# B&R Automation Studio project TD52 (part 149)

#### OpcHC.st
```iecst
(*******************************************************************************
OpcHC	 Variables read or write to Testbench

This code is confidential AND proprietary to the INNIO Company.
It may NOT be used in any form, or reproduced in any manner, without the express
written permission of the INNIO Company.
Copyright, INNIO Company, 2022

- list addidtional customized IO channels

Customized modifications: -
------------------------

History:
-------
V1.00.0	14.09.2022		Vockenberger	Neu erstellt
V1.01.0	31.05.2023		Vockenberger	Diff-Drucküberwachung Kühler mit Parameter
		28.07.2023		Vockenberger	Struktur von OPC_DI geändert
V1.02.0	20.03.2024		Vockenberger	Heizhaus und V-Kühler Variablen hinzugefügt
V1.03.0	09.01.2025		Gruber St.		cleanUp after change of parameter structure

Instructions FOR use:
--------------------

Outstandings:
------------

*******************************************************************************)

PROGRAM _CYCLIC

	(**Wird von Motor-CPU geschrieben**********************)
	(**REAL**)
	(*Regler*)
	rOpcHC_R[0]	:=	VIS2MM.tCtr_ChCW_LT_In.Y_man;
	rOpcHC_R[1]	:=	VIS2MM.tCtr_ChCW_LT_In.X_min;
	rOpcHC_R[2]	:=	VIS2MM.tCtr_ChCW_LT_In.X_max;
	rOpcHC_R[3]	:=	INT_TO_REAL(VIS2MM.tCtr_ChCW_LT_In.Tune_quality);

	rOpcHC_R[4]	:=	VIS2MM.tCtr_ChCW_HT_In.Y_man;
	rOpcHC_R[5]	:=	VIS2MM.tCtr_ChCW_HT_In.X_min;
	rOpcHC_R[6]	:=	VIS2MM.tCtr_ChCW_HT_In.X_max;
	rOpcHC_R[7]	:=	INT_TO_REAL(VIS2MM.tCtr_ChCW_HT_In.Tune_quality);

	rOpcHC_R[8]		:=	VIS2MM.tCtr_ChCW_HT_LP_In.Y_man;
	rOpcHC_R[9]		:=	VIS2MM.tCtr_ChCW_HT_LP_In.X_min;
	rOpcHC_R[10]	:=	VIS2MM.tCtr_ChCW_HT_LP_In.X_max;
	rOpcHC_R[11]	:=	INT_TO_REAL(VIS2MM.tCtr_ChCW_HT_LP_In.Tune_quality);

	rOpcHC_R[12]	:=	VIS2MM.tCtr_ChCW_HT_HP_In.Y_man;
	rOpcHC_R[13]	:=	VIS2MM.tCtr_ChCW_HT_HP_In.X_min;
	rOpcHC_R[14]	:=	VIS2MM.tCtr_ChCW_HT_HP_In.X_max;
	rOpcHC_R[15]	:=	INT_TO_REAL(VIS2MM.tCtr_ChCW_HT_HP_In.Tune_quality);

	rOpcHC_R[16]	:=	VIS2MM.tCtr_ChCW_LT_LP_In.Y_man;
	rOpcHC_R[17]	:=	VIS2MM.tCtr_ChCW_LT_LP_In.X_min;
	rOpcHC_R[18]	:=	VIS2MM.tCtr_ChCW_LT_LP_In.X_max;
	rOpcHC_R[19]	:=	INT_TO_REAL(VIS2MM.tCtr_ChCW_LT_LP_In.Tune_quality);

	rOpcHC_R[20]	:=	VIS2MM.tCtr_ChCW_LT_HP_In.Y_man;
	rOpcHC_R[21]	:=	VIS2MM.tCtr_ChCW_LT_HP_In.X_min;
	rOpcHC_R[22]	:=	VIS2MM.tCtr_ChCW_LT_HP_In.X_max;
	rOpcHC_R[23]	:=	INT_TO_REAL(VIS2MM.tCtr_ChCW_LT_HP_In.Tune_quality);

	rOpcHC_R[24]	:=	VIS2MM.tCtr_ECW_In.Y_man;
	rOpcHC_R[25]	:=	VIS2MM.tCtr_ECW_In.X_min;
	rOpcHC_R[26]	:=	VIS2MM.tCtr_ECW_In.X_max;
	rOpcHC_R[27]	:=	INT_TO_REAL(VIS2MM.tCtr_ECW_In.Tune_quality);

	rOpcHC_R[28]	:=	VIS2MM.tCtr_OCW_In.Y_man;
	rOpcHC_R[29]	:=	VIS2MM.tCtr_OCW_In.X_min;
	rOpcHC_R[30]	:=	VIS2MM.tCtr_OCW_In.X_max;
	rOpcHC_R[31]	:=	INT_TO_REAL(VIS2MM.tCtr_OCW_In.Tune_quality);

	rOpcHC_R[32]	:=	VIS2MM.tCtr_ChCW_LT_In.Y_set;
	rOpcHC_R[33]	:=	VIS2MM.tCtr_ChCW_HT_In.Y_set;
	rOpcHC_R[34]	:=	VIS2MM.tCtr_ChCW_LT_LP_In.Y_set;
	rOpcHC_R[35]	:=	VIS2MM.tCtr_ChCW_LT_HP_In.Y_set;
	rOpcHC_R[36]	:=	VIS2MM.tCtr_ChCW_HT_LP_In.Y_set;
	rOpcHC_R[37]	:=	VIS2MM.tCtr_ChCW_HT_HP_In.Y_set;
	rOpcHC_R[38]	:=	VIS2MM.tCtr_ECW_In.Y_set;
	rOpcHC_R[39]	:=	VIS2MM.tCtr_OCW_In.Y_set;

	rOpcHC_R[40]	:=	VIS2MM.rCtr_RW_CV_Set;
	rOpcHC_R[41]	:=	VIS2MM.rCtr_RW_HE_Set;
	rOpcHC_R[42]	:=	VIS2MM.rFC_ChCW_LT_PuSet;
	rOpcHC_R[43]	:=	VIS2MM.rFC_ChCW_HT_PuSet;
	rOpcHC_R[44]	:=	VIS2MM.rFC_ChCW_LT_LP_PuSet;
	rOpcHC_R[45]	:=	VIS2MM.rFC_ChCW_LT_HP_PuSet;
	rOpcHC_R[46]	:=	VIS2MM.rFC_ChCW_HT_LP_PuSet;
	rOpcHC_R[47]	:=	VIS2MM.rFC_ChCW_HT_HP_PuSet;
	rOpcHC_R[48]	:=	VIS2MM.rCtr_RW_LT_1_Set;
	rOpcHC_R[49]	:=	VIS2MM.rFC_ECW_PuSet;
	rOpcHC_R[50]	:=	VIS2MM.rFC_OCW_PuSet;

	rOpcHC_R[51]	:=	VIS2MM.rCtr_RW_HT_1_Set;
	rOpcHC_R[52]	:=	VIS2MM.rCtr_RW_LT_2_Set;
	rOpcHC_R[53]	:=	VIS2MM.rCtr_RW_HT_2_Set;
	rOpcHC_R[54]	:=	VIS2MM.rCtr_RW_ECW_1_Set;
	rOpcHC_R[55]	:=	VIS2MM.rCtr_RW_OCW_1_Set;
	rOpcHC_R[56]	:=	VIS2MM.rCtr_RW_ECW_2_Set;
	rOpcHC_R[57]	:=	VIS2MM.rCtr_RW_OCW_2_Set;
	rOpcHC_R[58]	:=	IN_DI.tT_HW_ReBeEng.Ai;

	rOpcHC_R[59]	:=	Para.tCtr_ECW.W_set;
	rOpcHC_R[60]	:=	Para.tCtr_OCW.W_set;
	rOpcHC_R[61]	:= 	Para.tCtr_ChCW_LT.W_set;
	rOpcHC_R[62]	:=	Para.tCtr_ChCW_LT_LP.W_set;
	rOpcHC_R[63]	:=	Para.tCtr_ChCW_LT_HP.W_set;
	rOpcHC_R[64]	:=	Para.tCtr_ChCW_HT.W_set;
	rOpcHC_R[65]	:=	Para.tCtr_ChCW_HT_LP.W_set;
	rOpcHC_R[66]	:=	Para.tCtr_ChCW_HT_HP.W_set;

	rOpcHC_R[67]	:=	Para.tCtr_ECW.W_min;
	rOpcHC_R[68]	:=	Para.tCtr_ECW.W_max;
	rOpcHC_R[69]	:=	Para.tCtr_ECW.Y_min;
	rOpcHC_R[70]	:=	Para.tCtr_ECW.Y_max;
	rOpcHC_R[71]	:=	Para.tCtr_OCW.W_min;
	rOpcHC_R[72]	:=	Para.tCtr_OCW.W_max;
	rOpcHC_R[73]	:=	Para.tCtr_OCW.Y_min;
	rOpcHC_R[74]	:=	Para.tCtr_OCW.Y_max;

	rOpcHC_R[75]	:=	Para.tCtr_ChCW_LT.W_min;
	rOpcHC_R[76]	:=	Para.tCtr_ChCW_LT.W_max;
	rOpcHC_R[77]	:=	Para.tCtr_ChCW_LT.Y_min;
	rOpcHC_R[78]	:=	Para.tCtr_ChCW_LT.Y_max;
	rOpcHC_R[79]	:=	Para.tCtr_ChCW_LT_LP.W_min;
	rOpcHC_R[80]	:=	Para.tCtr_ChCW_LT_LP.W_max;
	rOpcHC_R[81]	:=	Para.tCtr_ChCW_LT_LP.Y_min;
	rOpcHC_R[82]	:=	Para.tCtr_ChCW_LT_LP.Y_max;

	rOpcHC_R[83]	:=	Para.tCtr_ChCW_LT_HP.W_min;
	rOpcHC_R[84]	:=	Para.tCtr_ChCW_LT_HP.W_max;
	rOpcHC_R[85]	:=	Para.tCtr_ChCW_LT_HP.Y_min;
	rOpcHC_R[86]	:=	Para.tCtr_ChCW_LT_HP.Y_max;
	rOpcHC_R[87]	:=	Para.tCtr_ChCW_HT.W_min;
	rOpcHC_R[88]	:=	Para.tCtr_ChCW_HT.W_max;
	rOpcHC_R[89]	:=	Para.tCtr_ChCW_HT.Y_min;
	rOpcHC_R[90]	:=	Para.tCtr_ChCW_HT.Y_max;

	rOpcHC_R[91]	:=	Para.tCtr_ChCW_HT_LP.W_min;
	rOpcHC_R[92]	:=	Para.tCtr_ChCW_HT_LP.W_max;
	rOpcHC_R[93]	:=	Para.tCtr_ChCW_HT_LP.Y_min;
	rOpcHC_R[94]	:=	Para.tCtr_ChCW_HT_LP.Y_max;
	rOpcHC_R[95]	:=	Para.tCtr_ChCW_HT_HP.W_min;
	rOpcHC_R[96]	:=	Para.tCtr_ChCW_HT_HP.W_max;
	rOpcHC_R[97]	:=	Para.tCtr_ChCW_HT_HP.Y_min;
	rOpcHC_R[98]	:=	Para.tCtr_ChCW_HT_HP.Y_max;

	rOpcHC_R[99]	:=	VIS2MM.tPreHeatWDayLT[0].Hour;
	rOpcHC_R[100]	:=	VIS2MM.tPreHeatWDayLT[0].Minute;
	rOpcHC_R[101]	:=	VIS2MM.tPreHeatWDayLT[1].Hour;
	rOpcHC_R[102]	:=	VIS2MM.tPreHeatWDayLT[1].Minute;
	rOpcHC_R[103]	:=	VIS2MM.tPreHeatWDayLT[2].Hour;
	rOpcHC_R[104]	:=	VIS2MM.tPreHeatWDayLT[2].Minute;
	rOpcHC_R[105]	:=	VIS2MM.tPreHeatWDayLT[3].Hour;
	rOpcHC_R[106]	:=	VIS2MM.tPreHeatWDayLT[3].Minute;
	rOpcHC_R[107]	:=	VIS2MM.tPreHeatWDayLT[4].Hour;
	rOpcHC_R[108]	:=	VIS2MM.tPreHeatWDayLT[4].Minute;
	rOpcHC_R[109]	:=	VIS2MM.tPreHeatWDayLT[5].Hour;
	rOpcHC_R[110]	:=	VIS2MM.tPreHeatWDayLT[5].Minute;
	rOpcHC_R[111]	:=	VIS2MM.tPreHeatWDayLT[6].Hour;
	rOpcHC_R[112]	:=	VIS2MM.tPreHeatWDayLT[6].Minute;

	rOpcHC_R[113]	:=	VIS2MM.rT_LT_HP_Preh;
	rOpcHC_R[114]	:=	VIS2MM.rT_LT_LP_Preh;

	rOpcHC_R[115]	:=	IN_DI.tT_Ch_T2LP_A.Ai;
	rOpcHC_R[116]	:=	IN_DI.tT_Ch_T2LP_B.Ai;

	(**BOOL**)
	bOpcHC_R[0]  := VIS2MM.tCtr_ChCW_LT_In.Y_man_Active;
	bOpcHC_R[1]  := VIS2MM.tCtr_ChCW_LT_In.W_ext_Active;
	bOpcHC_R[2]  := VIS2MM.tCtr_ChCW_LT_In.Tune_PI;
	bOpcHC_R[3]  := VIS2MM.tCtr_ChCW_LT_In.Tune_PID;
	bOpcHC_R[4]  := VIS2MM.tCtr_ChCW_LT_In.Tune_start;
	bOpcHC_R[5]  := VIS2MM.tCtr_ChCW_LT_In.Tune_stop;
	bOpcHC_R[6]  := VIS2MM.tCtr_ChCW_LT_In.Tune_takeover;
	bOpcHC_R[7]	 := VIS2MM.tCtr_ChCW_LT_In.W_set2_Active;

	bOpcHC_R[8]   := VIS2MM.tCtr_ChCW_HT_In.Y_man_Active;
	bOpcHC_R[9]   := VIS2MM.tCtr_ChCW_HT_In.W_ext_Active;
	bOpcHC_R[10]  := VIS2MM.tCtr_ChCW_HT_In.Tune_PI;
	bOpcHC_R[11]  := VIS2MM.tCtr_ChCW_HT_In.Tune_PID;
	bOpcHC_R[12]  := VIS2MM.tCtr_ChCW_HT_In.Tune_start;
	bOpcHC_R[13]  := VIS2MM.tCtr_ChCW_HT_In.Tune_stop;
	bOpcHC_R[14]  := VIS2MM.tCtr_ChCW_HT_In.Tune_takeover;
	bOpcHC_R[15]  := VIS2MM.tCtr_ChCW_HT_In.W_set2_Active;

	bOpcHC_R[16]  := VIS2MM.tCtr_ChCW_HT_LP_In.Y_man_Active;
	bOpcHC_R[17]  := VIS2MM.tCtr_ChCW_HT_LP_In.W_ext_Active;
	bOpcHC_R[18]  := VIS2MM.tCtr_ChCW_HT_LP_In.Tune_PI;
	bOpcHC_R[19]  := VIS2MM.tCtr_ChCW_HT_LP_In.Tune_PID;
	bOpcHC_R[20]  := VIS2MM.tCtr_ChCW_HT_LP_In.Tune_start;
	bOpcHC_R[21]  := VIS2MM.tCtr_ChCW_HT_LP_In.Tune_stop;
	bOpcHC_R[22]  := VIS2MM.tCtr_ChCW_HT_LP_In.Tune_takeover;
	bOpcHC_R[23]  := VIS2MM.tCtr_ChCW_HT_LP_In.W_set2_Active;

	bOpcHC_R[24]  := VIS2MM.tCtr_ChCW_HT_HP_In.Y_man_Active;
	bOpcHC_R[25]  := VIS2MM.tCtr_ChCW_HT_HP_In.W_ext_Active;
	bOpcHC_R[26]  := VIS2MM.tCtr_ChCW_HT_HP_In.Tune_PI;
	bOpcHC_R[27]  := VIS2MM.tCtr_ChCW_HT_HP_In.Tune_PID;
	bOpcHC_R[28]  := VIS2MM.tCtr_ChCW_HT_HP_In.Tune_start;
	bOpcHC_R[29]  := VIS2MM.tCtr_ChCW_HT_HP_In.Tune_stop;
	bOpcHC_R[30]  := VIS2MM.tCtr_ChCW_HT_HP_In.Tune_takeover;
	bOpcHC_R[31]  := VIS2MM.tCtr_ChCW_HT_HP_In.W_set2_Active;

	bOpcHC_R[32]  := VIS2MM.tCtr_ChCW_LT_LP_In.Y_man_Active;
	bOpcHC_R[33]  := VIS2MM.tCtr_ChCW_LT_LP_In.W_ext_Active;
	bOpcHC_R[34]  := VIS2MM.tCtr_ChCW_LT_LP_In.Tune_PI;
	bOpcHC_R[35]  := VIS2MM.tCtr_ChCW_LT_LP_In.Tune_PID;
	bOpcHC_R[36]  := VIS2MM.tCtr_ChCW_LT_LP_In.Tune_start;
	bOpcHC_R[37]  := VIS2MM.tCtr_ChCW_LT_LP_In.Tune_stop;
	bOpcHC_R[38]  := VIS2MM.tCtr_ChCW_LT_LP_In.Tune_takeover;
	bOpcHC_R[39]  := VIS2MM.tCtr_ChCW_LT_LP_In.W_set2_Active;

	bOpcHC_R[40]  := VIS2MM.tCtr_ChCW_LT_HP_In.Y_man_Active;
	bOpcHC_R[41]  := VIS2MM.tCtr_ChCW_LT_HP_In.W_ext_Active;
	bOpcHC_R[42]  := VIS2MM.tCtr_ChCW_LT_HP_In.Tune_PI;
	bOpcHC_R[43]  := VIS2MM.tCtr_ChCW_LT_HP_In.Tune_PID;
	bOpcHC_R[44]  := VIS2MM.tCtr_ChCW_LT_HP_In.Tune_start;
	bOpcHC_R[45]  := VIS2MM.tCtr_ChCW_LT_HP_In.Tune_stop;
	bOpcHC_R[46]  := VIS2MM.tCtr_ChCW_LT_HP_In.Tune_takeover;
	bOpcHC_R[47]  := VIS2MM.tCtr_ChCW_LT_HP_In.W_set2_Active;

	bOpcHC_R[48]  := VIS2MM.tCtr_ECW_In.Y_man_Active;
	bOpcHC_R[49]  := VIS2MM.tCtr_ECW_In.W_ext_Active;
	bOpcHC_R[50]  := VIS2MM.tCtr_ECW_In.Tune_PI;
	bOpcHC_R[51]  := VIS2MM.tCtr_ECW_In.Tune_PID;
	bOpcHC_R[52]  := VIS2MM.tCtr_ECW_In.Tune_start;
	bOpcHC_R[53]  := VIS2MM.tCtr_ECW_In.Tune_stop;
	bOpcHC_R[54]  := VIS2MM.tCtr_ECW_In.Tune_takeover;
	bOpcHC_R[55]  := VIS2MM.tCtr_ECW_In.W_set2_Active;

	bOpcHC_R[56]  := VIS2MM.tCtr_OCW_In.Y_man_Active;
	bOpcHC_R[57]  := VIS2MM.tCtr_OCW_In.W_ext_Active;
	bOpcHC_R[58]  := VIS2MM.tCtr_OCW_In.Tune_PI;
	bOpcHC_R[59]  := VIS2MM.tCtr_OCW_In.Tune_PID;
	bOpcHC_R[60]  := VIS2MM.tCtr_OCW_In.Tune_start;
	bOpcHC_R[61]  := VIS2MM.tCtr_OCW_In.Tune_stop;
	bOpcHC_R[62]  := VIS2MM.tCtr_OCW_In.Tune_takeover;
	bOpcHC_R[63]  := VIS2MM.tCtr_OCW_In.W_set2_Active;

	bOpcHC_R[64]  := bCtr_LT_In_Y_set_Active;
	bOpcHC_R[65]  := bCtr_HT_In_Y_set_Active;
	bOpcHC_R[66]  := bCtr_LT_LP_In_Y_set_Active;
	bOpcHC_R[67]  := bCtr_LT_HP_In_Y_set_Active;
	bOpcHC_R[68]  := bCtr_HT_LP_In_Y_set_Active;
	bOpcHC_R[69]  := bCtr_HT_HP_In_Y_set_Active;
	bOpcHC_R[70]  := bCtr_ECW_In_Y_set_Active;
	bOpcHC_R[71]  := bCtr_OCW_In_Y_set_Active;

	bOpcHC_R[72]  := VIS2MM.bMan_ECW_Pump;
	bOpcHC_R[73]  := VIS2MM.bMan_OCW_Pump;
	bOpcHC_R[74]  := VIS2MM.bMan_LT_Pump;
	bOpcHC_R[75]  := VIS2MM.bMan_HT_Pump;
	bOpcHC_R[76]  := VIS2MM.bMan_LT_LP_Pump;
	bOpcHC_R[77]  := VIS2MM.bMan_LT_HP_Pump;
	bOpcHC_R[78]  := VIS2MM.bMan_HT_LP_Pump;
	bOpcHC_R[79]  := VIS2MM.bMan_HT_HP_Pump;

	bOpcHC_R[80]	:=	VIS2MM.bMan_BoilerHouse_Pump;
	bOpcHC_R[81]	:=	VIS2MM.bMan_SecCirc_Pump;
	bOpcHC_R[82]	:=	VIS2MM.bPreHeatWDayLT_CtrActive;
	bOpcHC_R[83]	:=	VIS2MM.bLT_PreH_Dem;
	bOpcHC_R[84]	:=	VIS2MM.tPreHeatWDayLT[0].Active;
	bOpcHC_R[85]	:=	VIS2MM.tPreHeatWDayLT[1].Active;
	bOpcHC_R[86]	:=	VIS2MM.tPreHeatWDayLT[2].Active;
	bOpcHC_R[87]	:=	VIS2MM.tPreHeatWDayLT[3].Active;
	bOpcHC_R[88]	:=	VIS2MM.tPreHeatWDayLT[4].Active;
	bOpcHC_R[89]	:=	VIS2MM.tPreHeatWDayLT[5].Active;
	bOpcHC_R[90]	:=	VIS2MM.tPreHeatWDayLT[6].Active;
	bOpcHC_R[91]	:=	VIS2MM.tPreHeatWDayLT[7].Active;
	bOpcHC_R[92]	:=	VIS2MM.tPreHeatWDayLT[0].Off;
	bOpcHC_R[93]	:=	VIS2MM.tPreHeatWDayLT[1].Off;
	bOpcHC_R[94]	:=	VIS2MM.tPreHeatWDayLT[2].Off;
	bOpcHC_R[95]	:=	VIS2MM.tPreHeatWDayLT[3].Off;
	bOpcHC_R[96]	:=	VIS2MM.tPreHeatWDayLT[4].Off;
	bOpcHC_R[97]	:=	VIS2MM.tPreHeatWDayLT[5].Off;
	bOpcHC_R[98]	:=	VIS2MM.tPreHeatWDayLT[6].Off;
	bOpcHC_R[99]	:=	IN_DI.tT_Ch_T2LP_A.Exist;
	bOpcHC_R[100];

	(**Wird von Prüfstands-CPU geschrieben**********************)
	(**REAL**)
	MM2VIS.rT_ChCW_Re_LT		:=	rOpcHC_W[0];
	MM2VIS.rPr_ChCW_Re_LT		:=	rOpcHC_W[1];
	MM2VIS.rT_ChCW_Su_LT		:=	rOpcHC_W[2];
	MM2VIS.rPr_ChCW_Su_LT		:=	rOpcHC_W[3];
	MM2VIS.rT_ChCW_Re_HT		:=	rOpcHC_W[4];
	MM2VIS.rPr_ChCW_Re_HT		:=	rOpcHC_W[5];
	MM2VIS.rT_ChCW_Su_HT		:=	rOpcHC_W[6];
	MM2VIS.rPr_ChCW_Su_HT		:=	rOpcHC_W[7];
	MM2VIS.rT_ChCW_Re_HT_LP		:=	rOpcHC_W[8];
	MM2VIS.rPr_ChCW_Re_HT_LP	:=	rOpcHC_W[9];

	MM2VIS.rT_ChCW_Re_HT_HP		:=	rOpcHC_W[10];
	MM2VIS.rPr_ChCW_Re_HT_HP	:=	rOpcHC_W[11];
	MM2VIS.rT_ChCW_Su_HT_LP		:=	rOpcHC_W[12];
	MM2VIS.rPr_ChCW_Su_HT_LP	:=	rOpcHC_W[13];
	MM2VIS.rT_ChCW_Su_HT_HP		:=	rOpcHC_W[14];
	MM2VIS.rPr_ChCW_Su_HT_HP	:=	rOpcHC_W[15];
	MM2VIS.rT_ChCW_Re_LT_LP		:=	rOpcHC_W[16];
	MM2VIS.rPr_ChCW_Re_LT_LP	:=	rOpcHC_W[17];
	MM2VIS.rT_ChCW_Re_LT_HP		:=	rOpcHC_W[18];
	MM2VIS.rPr_ChCW_Re_LT_HP	:=	rOpcHC_W[19];

	MM2VIS.rT_ChCW_Su_LT_LP		:=	rOpcHC_W[20];
	MM2VIS.rPr_ChCW_Su_LT_LP	:=	rOpcHC_W[21];
	MM2VIS.rT_ChCW_Su_LT_HP		:=	rOpcHC_W[22];
	MM2VIS.rPr_ChCW_Su_LT_HP	:=	rOpcHC_W[23];
	MM2VIS.rT_OCW_Re			:=	rOpcHC_W[24];
	MM2VIS.rPr_OCW_Re			:=	rOpcHC_W[25];
	MM2VIS.rT_OCW_Su			:=	rOpcHC_W[26];
	MM2VIS.rPr_OCW_Su			:=	rOpcHC_W[27];
	MM2VIS.rT_ECW_Re			:=	rOpcHC_W[28];
	MM2VIS.rPr_ECW_Re			:=	rOpcHC_W[29];

	MM2VIS.rT_ECW_Su			:=	rOpcHC_W[30];
	MM2VIS.rPr_ECW_Su			:=	rOpcHC_W[31];
	MM2VIS.rVol_ChCW_Re_LT		:=	rOpcHC_W[32];
	MM2VIS.rVol_ChCW_Su_LT		:=	rOpcHC_W[33];
	MM2VIS.rVol_ChCW_Re_HT		:=	rOpcHC_W[34];
	MM2VIS.rVol_ChCW_Su_HT		:=	rOpcHC_W[35];
	MM2VIS.rVol_ChCW_Re_HT_LP	:=	rOpcHC_W[36];
	MM2VIS.rVol_ChCW_Su_HT_LP	:=	rOpcHC_W[37];
	MM2VIS.rVol_ChCW_Re_HT_HP	:=	rOpcHC_W[38];
	MM2VIS.rVol_ChCW_Su_HT_HP	:=	rOpcHC_W[39];

	MM2VIS.rVol_ChCW_Re_LT_LP	:=	rOpcHC_W[40];
	MM2VIS.rVol_ChCW_Su_LT_LP	:=	rOpcHC_W[41];
	MM2VIS.rVol_ChCW_Re_LT_HP	:=	rOpcHC_W[42];
	MM2VIS.rVol_ChCW_Su_LT_HP	:=	rOpcHC_W[43];
	MM2VIS.rVol_ECW_Re			:=	rOpcHC_W[44];
	MM2VIS.rVol_ECW_Su			:=	rOpcHC_W[45];
	MM2VIS.rVol_OCW_Re			:=	rOpcHC_W[46];
	MM2VIS.rVol_OCW_Su			:=	rOpcHC_W[47];
	MM2VIS.rPosAct_RW_LT_1		:=	rOpcHC_W[48];
	MM2VIS.rPosAct_RW_HT_1		:=	rOpcHC_W[49];

	MM2VIS.rT_ChCW_LT_IC_Re		:=	rOpcHC_W[50];
	MM2VIS.rPr_ChCW_LT_IC_Re	:=	rOpcHC_W[51];
	MM2VIS.rT_ChCW_HT_IC_Re		:=	rOpcHC_W[52];
	MM2VIS.rPr_ChCW_HT_IC_Re	:=	rOpcHC_W[53];
	MM2VIS.rT_ChCW_LT_LP_IC_Re	:=	rOpcHC_W[54];
	MM2VIS.rPr_ChCW_LT_LP_IC_Re	:=	rOpcHC_W[55];
	MM2VIS.rT_ChCW_LT_HP_IC_Re	:=	rOpcHC_W[56];
	MM2VIS.rPr_ChCW_LT_HP_IC_Re	:=	rOpcHC_W[57];
	MM2VIS.rT_ChCW_HT_LP_IC_Re	:=	rOpcHC_W[58];
	MM2VIS.rPr_ChCW_HT_LP_IC_Re	:=	rOpcHC_W[59];

	MM2VIS.rT_ChCW_HT_HP_IC_Re	:=	rOpcHC_W[60];
	MM2VIS.rPr_ChCW_HT_HP_IC_Re	:=	rOpcHC_W[61];
	MM2VIS.rT_RW_Re				:=	rOpcHC_W[62];
	MM2VIS.rT_RW_Su				:=	rOpcHC_W[63];
	MM2VIS.rT_ECW_IC_Re			:=	rOpcHC_W[64];
	MM2VIS.rPr_ECW_IC_Re		:=	rOpcHC_W[65];
	MM2VIS.rT_OCW_IC_Re			:=	rOpcHC_W[66];
	MM2VIS.rPr_OCW_IC_Re		:=	rOpcHC_W[67];
	MM2VIS.rT_ChCW_LT_IC_Su		:=	rOpcHC_W[68];
	MM2VIS.rPr_ChCW_LT_IC_Su	:=	rOpcHC_W[69];

	MM2VIS.rT_ChCW_HT_IC_Su		:=	rOpcHC_W[70];
	MM2VIS.rPr_ChCW_HT_IC_Su	:=	rOpcHC_W[71];
	MM2VIS.rT_ChCW_LT_LP_IC_Su	:=	rOpcHC_W[72];
	MM2VIS.rPr_ChCW_LT_LP_IC_Su	:=	rOpcHC_W[73];
	MM2VIS.rT_ChCW_LT_HP_IC_Su	:=	rOpcHC_W[74];
	MM2VIS.rPr_ChCW_LT_HP_IC_Su	:=	rOpcHC_W[75];
	MM2VIS.rT_ChCW_HT_LP_IC_Su	:=	rOpcHC_W[76];
	MM2VIS.rPr_ChCW_HT_LP_IC_Su	:=	rOpcHC_W[77];
	MM2VIS.rT_ChCW_HT_HP_IC_Su	:=	rOpcHC_W[78];
	MM2VIS.rPr_ChCW_HT_HP_IC_Su	:=	rOpcHC_W[79];

	MM2VIS.rPr_RW_LT_Re_1		:=	rOpcHC_W[80];
	MM2VIS.rPr_RW_LT_Su_1		:=	rOpcHC_W[81];
	MM2VIS.rT_ECW_IC_Su			:=	rOpcHC_W[82];
	MM2VIS.rPr_ECW_IC_Su		:=	rOpcHC_W[83];
	MM2VIS.rT_OCW_IC_Su			:=	rOpcHC_W[84];
	MM2VIS.rPr_OCW_IC_Su		:=	rOpcHC_W[85];
	MM2VIS.rT_Cooler_ChCW_LT_Re_1	:=	rOpcHC_W[86];
	MM2VIS.rT_Cooler_ChCW_HT_Re_1	:=	rOpcHC_W[87];
	MM2VIS.rT_Cooler_ChCW_HT_Re_3	:=	rOpcHC_W[88];
	MM2VIS.rT_Cooler_ChCW_HT_Re_4	:=	rOpcHC_W[89];

	MM2VIS.rT_Cooler_ChCW_HT_Re_5	:=	rOpcHC_W[90];
	MM2VIS.rT_Cooler_ChCW_HT_Su_3	:=	rOpcHC_W[91];
	MM2VIS.rT_Cooler_ChCW_LT_Re_2		:=	rOpcHC_W[92];
	MM2VIS.rT_Cooler_ChCW_HT_Re_2		:=	rOpcHC_W[93];
	MM2VIS.rT_Cooler_ChCW_HT_Su_4	:=	rOpcHC_W[94];
	MM2VIS.rT_Cooler_ChCW_HT_Su_5	:=	rOpcHC_W[95];
	MM2VIS.rT_CoolerCabinet_HT_1	:=	rOpcHC_W[96];
	MM2VIS.rT_CoolerCabinet_HT_2	:=	rOpcHC_W[97];
	MM2VIS.rPr_Cooler_ChCW_LT_Re_1		:=	rOpcHC_W[98];
	MM2VIS.rPr_Cooler_ChCW_HT_Re_1		:=	rOpcHC_W[99];

	MM2VIS.rT_CoolerCabinet_HT_3		:=	rOpcHC_W[100];
	MM2VIS.rT_CoolerCabinet_HT_4		:=	rOpcHC_W[101];
	MM2VIS.rT_CoolerCabinet_HT_5		:=	rOpcHC_W[102];
	MM2VIS.rT_Cooler_OCW_Re_3			:=	rOpcHC_W[103];
	MM2VIS.rPr_Cooler_ChCW_LT_Re_2		:=	rOpcHC_W[104];
	MM2VIS.rPr_Cooler_ChCW_HT_Re_2		:=	rOpcHC_W[105];
	MM2VIS.rT_Cooler_OCW_Su_3			:=	rOpcHC_W[106];
	MM2VIS.rT_CoolerCabinet_OCW_1		:=	rOpcHC_W[107];
	MM2VIS.rT_CoolerCabinet_OCW_2		:=	rOpcHC_W[108];
	MM2VIS.rT_CoolerCabinet_OCW_3		:=	rOpcHC_W[109];

	MM2VIS.rT_Cooler_ChCW_LT_Su_1		:=	rOpcHC_W[110];
	MM2VIS.rT_Cooler_ChCW_HT_Su_1		:=	rOpcHC_W[111];
	MM2VIS.rT_Cooler_ECW_Re_3			:=	rOpcHC_W[112];
	MM2VIS.rT_Cooler_ECW_Re_4			:=	rOpcHC_W[113];
	MM2VIS.rT_Cooler_ECW_Su_3			:=	rOpcHC_W[114];
	MM2VIS.rT_Cooler_ECW_Su_4			:=	rOpcHC_W[115];
	MM2VIS.rT_Cooler_ChCW_LT_Su_2		:=	rOpcHC_W[116];
	MM2VIS.rT_Cooler_ChCW_HT_Su_2		:=	rOpcHC_W[117];
	MM2VIS.rT_CoolerCabinet_ECW_1		:=	rOpcHC_W[118];
	MM2VIS.rT_CoolerCabinet_ECW_2		:=	rOpcHC_W[119];

	MM2VIS.rT_CoolerCabinet_ECW_3		:=	rOpcHC_W[120];
	MM2VIS.rT_CoolerCabinet_ECW_4		:=	rOpcHC_W[121];
	MM2VIS.rPr_Cooler_ChCW_LT_Su_1		:=	rOpcHC_W[122];
	MM2VIS.rPr_Cooler_ChCW_HT_Su_1		:=	rOpcHC_W[123];
	MM2VIS.rT_Cooler_ChCW_LT_Re_3		:=	rOpcHC_W[124];
	MM2VIS.rT_Cooler_ChCW_LT_Re_4		:=	rOpcHC_W[125];
	MM2VIS.rT_Cooler_ChCW_LT_Re_5		:=	rOpcHC_W[126];
	MM2VIS.rT_Cooler_ChCW_LT_Su_3		:=	rOpcHC_W[127];
	MM2VIS.rPr_Cooler_ChCW_LT_Su_2		:=	rOpcHC_W[128];
	MM2VIS.rPr_Cooler_ChCW_HT_Su_2		:=	rOpcHC_W[129];

	MM2VIS.rT_Cooler_ChCW_LT_Su_4	:=	rOpcHC_W[130];
	MM2VIS.rT_Cooler_ChCW_LT_Su_5	:=	rOpcHC_W[131];
	MM2VIS.rT_CoolerCabinet_LT_1	:=	rOpcHC_W[132];
	MM2VIS.rT_CoolerCabinet_LT_2	:=	rOpcHC_W[133];
	MM2VIS.rPr_RW_LT_Re_2		:=	rOpcHC_W[134];
	MM2VIS.rPr_RW_LT_Su_2		:=	rOpcHC_W[135];
	MM2VIS.rT_Cooler_ECW_Re_1	:=	rOpcHC_W[136];
	MM2VIS.rT_Cooler_ECW_Re_2	:=	rOpcHC_W[137];
	MM2VIS.rT_Cooler_OCW_Re_1	:=	rOpcHC_W[138];
	MM2VIS.rT_Cooler_OCW_Re_2	:=	rOpcHC_W[139];

	MM2VIS.rPr_RW_HT_Re_1		:=	rOpcHC_W[140];
	MM2VIS.rPr_RW_HT_Su_1		:=	rOpcHC_W[141];
	MM2VIS.rT_Cooler_ECW_Su_1	:=	rOpcHC_W[142];
	MM2VIS.rT_Cooler_ECW_Su_2	:=	rOpcHC_W[143];
	MM2VIS.rT_Cooler_OCW_Su_1	:=	rOpcHC_W[144];
	MM2VIS.rT_Cooler_OCW_Su_2	:=	rOpcHC_W[145];
	MM2VIS.rT_ChCW_LT_bCV		:=	rOpcHC_W[146];
	MM2VIS.rT_RW_HE_Re			:=	rOpcHC_W[147];
	MM2VIS.rT_RW_HE_Su			:=	rOpcHC_W[148];
	MM2VIS.rPr_RW_HT_Re_2		:=	rOpcHC_W[149];

	MM2VIS.rPr_RW_HT_Su_2		:=	rOpcHC_W[150];
	MM2VIS.rPr_Cooler_ECW_Re_1	:=	rOpcHC_W[151];
	MM2VIS.rPr_Cooler_ECW_Re_2	:=	rOpcHC_W[152];
	MM2VIS.rPr_Cooler_OCW_Re_1	:=	rOpcHC_W[153];
	MM2VIS.rPr_Cooler_OCW_Re_2	:=	rOpcHC_W[154];
	MM2VIS.rPr_RW_ECW_Re_1		:=	rOpcHC_W[155];
	MM2VIS.rPr_RW_ECW_Su_1		:=	rOpcHC_W[156];
	MM2VIS.rPr_Cooler_ECW_Su_1	:=	rOpcHC_W[157];
	MM2VIS.rPr_Cooler_ECW_Su_2	:=	rOpcHC_W[158];
	MM2VIS.rPr_Cooler_OCW_Su_1	:=	rOpcHC_W[159];

	MM2VIS.rPr_Cooler_OCW_Su_2	:=	rOpcHC_W[160];
	MM2VIS.rPr_RW_HE_Re			:=	rOpcHC_W[161];
	MM2VIS.rPr_RW_HE_Su			:=	rOpcHC_W[162];
	MM2VIS.rFC_ChCW_LT_Pump		:=	rOpcHC_W[163];
	MM2VIS.rFC_ChCW_HT_Pump		:=	rOpcHC_W[164];
	MM2VIS.rFC_ChCW_LT_LP_Pump	:=	rOpcHC_W[165];
	MM2VIS.rFC_ChCW_LT_HP_Pump	:=	rOpcHC_W[166];
	MM2VIS.rFC_ChCW_HT_LP_Pump	:=	rOpcHC_W[167];
	MM2VIS.rFC_ChCW_HT_HP_Pump	:=	rOpcHC_W[168];
	MM2VIS.rPr_RW_ECW_Re_2		:=	rOpcHC_W[169];

	MM2VIS.rFC_ECW_Pump			:=	rOpcHC_W[170];
	MM2VIS.rFC_OCW_Pump			:=	rOpcHC_W[171];
	MM2VIS.rFC_ChCW_LT_Cooler_1	:=	rOpcHC_W[172];
	MM2VIS.rFC_ChCW_HT_Cooler_1	:=	rOpcHC_W[173];
	MM2VIS.rT_CoolerCabinet_LT_3	:=	rOpcHC_W[174];
	MM2VIS.rT_CoolerCabinet_LT_4	:=	rOpcHC_W[175];
	MM2VIS.rT_CoolerCabinet_LT_5	:=	rOpcHC_W[176];
	MM2VIS.rFC_ChCW_HT_HP_Cooler_1	:=	rOpcHC_W[177];
	MM2VIS.rFC_ChCW_LT_Cooler_2	:=	rOpcHC_W[178];
	MM2VIS.rFC_ChCW_HT_Cooler_2	:=	rOpcHC_W[179];

	MM2VIS.rFC_ChCW_LT_LP_Cooler_2	:=	rOpcHC_W[180];
	MM2VIS.rFC_ChCW_LT_HP_Cooler_2	:=	rOpcHC_W[181];
	MM2VIS.rFC_ChCW_HT_LP_Cooler_2	:=	rOpcHC_W[182];
	MM2VIS.rFC_ChCW_HT_HP_Cooler_2	:=	rOpcHC_W[183];
	MM2VIS.rPr_RW_ECW_Su_2		:=	rOpcHC_W[184];
	MM2VIS.rFC_ECW_Cooler_1		:=	rOpcHC_W[185];
	MM2VIS.rFC_OCW_Cooler_1		:=	rOpcHC_W[186];
	MM2VIS.rPr_RW_OCW_Re_1		:=	rOpcHC_W[187];
	MM2VIS.rFC_ECW_Cooler_2		:=	rOpcHC_W[188];
	MM2VIS.rFC_OCW_Cooler_2		:=	rOpcHC_W[189];

	MM2VIS.rT_ChCW_LT_LP_bCV	:=	rOpcHC_W[190];
	MM2VIS.rT_ChCW_LT_HP_bCV	:=	rOpcHC_W[191];
	MM2VIS.rT_ChCW_HT_bCV		:=	rOpcHC_W[192];
	MM2VIS.rT_ChCW_HT_LP_bCV	:=	rOpcHC_W[193];
	MM2VIS.rT_ChCW_HT_HP_bCV	:=	rOpcHC_W[194];
	MM2VIS.rPr_RW_OCW_Su_1		:=	rOpcHC_W[195];
	MM2VIS.rT_ECW_bCV			:=	rOpcHC_W[196];
	MM2VIS.rT_OCW_bCV			:=	rOpcHC_W[197];
	MM2VIS.rPosAct_ChCW_LT		:=	rOpcHC_W[198];
	MM2VIS.rPosAct_ChCW_HT		:=	rOpcHC_W[199];

	MM2VIS.rPosAct_ChCW_HT_LP	:=	rOpcHC_W[200];
	MM2VIS.rPosAct_ChCW_HT_HP	:=	rOpcHC_W[201];
	MM2VIS.rPosAct_ChCW_LT_LP	:=	rOpcHC_W[202];
	MM2VIS.rPosAct_ChCW_LT_HP	:=	rOpcHC_W[203];
	MM2VIS.rPosAct_ECW			:=	rOpcHC_W[204];
	MM2VIS.rPosAct_OCW			:=	rOpcHC_W[205];
	MM2VIS.rPr_RW_OCW_Re_2		:=	rOpcHC_W[206];
	MM2VIS.rPosAct_RW_CV		:=	rOpcHC_W[207];
	MM2VIS.rPosAct_RW_HE		:=	rOpcHC_W[208];

	(**Regler**)
	MM2VIS.rCtr_ChCW_LT_In_X		:=	rOpcHC_W[209];
	MM2VIS.tCtr_ChCW_LT_Out.Y		:=	rOpcHC_W[210];
	MM2VIS.tCtr_ChCW_LT_Out.Y_min_act	:=	rOpcHC_W[211];
	MM2VIS.tCtr_ChCW_LT_Out.Y_max_act	:=	rOpcHC_W[212];
	MM2VIS.tCtr_ChCW_LT_Out.W		:=	rOpcHC_W[213];
	MM2VIS.tCtr_ChCW_LT_Out.e		:=	rOpcHC_W[214];
	MM2VIS.tCtr_ChCW_LT_Out.Kp_tune	:=	rOpcHC_W[215];
	MM2VIS.tCtr_ChCW_LT_Out.Tn_tune	:=	rOpcHC_W[216];
	MM2VIS.tCtr_ChCW_LT_Out.Tv_tune	:=	rOpcHC_W[217];
	MM2VIS.tCtr_ChCW_LT_Out.status	:=	REAL_TO_UINT(rOpcHC_W[218]);
	MM2VIS.tCtr_ChCW_LT_Out.Kp_act	:=	rOpcHC_W[219];
	MM2VIS.tCtr_ChCW_LT_Out.Tn_act	:=	rOpcHC_W[220];
	MM2VIS.tCtr_ChCW_LT_Out.Tv_act	:=	rOpcHC_W[221];

	MM2VIS.rCtr_ChCW_HT_In_X		:=	rOpcHC_W[222];
	MM2VIS.tCtr_ChCW_HT_Out.Y		:=	rOpcHC_W[223];
	MM2VIS.tCtr_ChCW_HT_Out.Y_min_act	:=	rOpcHC_W[224];
	MM2VIS.tCtr_ChCW_HT_Out.Y_max_act	:=	rOpcHC_W[225];
	MM2VIS.tCtr_ChCW_HT_Out.W		:=	rOpcHC_W[226];
	MM2VIS.tCtr_ChCW_HT_Out.e		:=	rOpcHC_W[227];
	MM2VIS.tCtr_ChCW_HT_Out.Kp_tune	:=	rOpcHC_W[228];
	MM2VIS.tCtr_ChCW_HT_Out.Tn_tune	:=	rOpcHC_W[229];
	MM2VIS.tCtr_ChCW_HT_Out.Tv_tune	:=	rOpcHC_W[230];
	MM2VIS.tCtr_ChCW_HT_Out.status	:=	REAL_TO_UINT(rOpcHC_W[231]);
	MM2VIS.tCtr_ChCW_HT_Out.Kp_act	:=	rOpcHC_W[232];
	MM2VIS.tCtr_ChCW_HT_Out.Tn_act	:=	rOpcHC_W[233];
	MM2VIS.tCtr_ChCW_HT_Out.Tv_act	:=	rOpcHC_W[234];

	MM2VIS.rCtr_ChCW_HT_LP_In_X			:=	rOpcHC_W[235];
	MM2VIS.tCtr_ChCW_HT_LP_Out.Y		:=	rOpcHC_W[236];
	MM2VIS.tCtr_ChCW_HT_LP_Out.Y_min_act	:=	rOpcHC_W[237];
	MM2VIS.tCtr_ChCW_HT_LP_Out.Y_max_act	:=	rOpcHC_W[238];
	MM2VIS.tCtr_ChCW_HT_LP_Out.W		:=	rOpcHC_W[239];
	MM2VIS.tCtr_ChCW_HT_LP_Out.e		:=	rOpcHC_W[240];
	MM2VIS.tCtr_ChCW_HT_LP_Out.Kp_tune	:=	rOpcHC_W[241];
	MM2VIS.tCtr_ChCW_HT_LP_Out.Tn_tune	:=	rOpcHC_W[242];
	MM2VIS.tCtr_ChCW_HT_LP_Out.Tv_tune	:=	rOpcHC_W[243];
	MM2VIS.tCtr_ChCW_HT_LP_Out.status	:=	REAL_TO_UINT(rOpcHC_W[244]);
	MM2VIS.tCtr_ChCW_HT_LP_Out.Kp_act	:=	rOpcHC_W[245];
	MM2VIS.tCtr_ChCW_HT_LP_Out.Tn_act	:=	rOpcHC_W[246];
	MM2VIS.tCtr_ChCW_HT_LP_Out.Tv_act	:=	rOpcHC_W[247];

	MM2VIS.rCtr_ChCW_HT_HP_In_X			:=	rOpcHC_W[248];
	MM2VIS.tCtr_ChCW_HT_HP_Out.Y		:=	rOpcHC_W[249];
	MM2VIS.tCtr_ChCW_HT_HP_Out.Y_min_act	:=	rOpcHC_W[250];
	MM2VIS.tCtr_ChCW_HT_HP_Out.Y_max_act	:=	rOpcHC_W[251];
	MM2VIS.tCtr_ChCW_HT_HP_Out.W		:=	rOpcHC_W[252];
	MM2VIS.tCtr_ChCW_HT_HP_Out.e		:=	rOpcHC_W[253];
	MM2VIS.tCtr_ChCW_HT_HP_Out.Kp_tune	:=	rOpcHC_W[254];
	MM2VIS.tCtr_ChCW_HT_HP_Out.Tn_tune	:=	rOpcHC_W[255];
	MM2VIS.tCtr_ChCW_HT_HP_Out.Tv_tune	:=	rOpcHC_W[256];
	MM2VIS.tCtr_ChCW_HT_HP_Out.status	:=	REAL_TO_UINT(rOpcHC_W[257]);
	MM2VIS.tCtr_ChCW_HT_HP_Out.Kp_act	:=	rOpcHC_W[258];
	MM2VIS.tCtr_ChCW_HT_HP_Out.Tn_act	:=	rOpcHC_W[259];
	MM2VIS.tCtr_ChCW_HT_HP_Out.Tv_act	:=	rOpcHC_W[260];

	MM2VIS.rCtr_ChCW_LT_LP_In_X			:=	rOpcHC_W[261];
	MM2VIS.tCtr_ChCW_LT_LP_Out.Y		:=	rOpcHC_W[262];
	MM2VIS.tCtr_ChCW_LT_LP_Out.Y_min_act	:=	rOpcHC_W[263];
	MM2VIS.tCtr_ChCW_LT_LP_Out.Y_max_act	:=	rOpcHC_W[264];
	MM2VIS.tCtr_ChCW_LT_LP_Out.W		:=	rOpcHC_W[265];
	MM2VIS.tCtr_ChCW_LT_LP_Out.e		:=	rOpcHC_W[266];
	MM2VIS.tCtr_ChCW_LT_LP_Out.Kp_tune	:=	rOpcHC_W[267];
	MM2VIS.tCtr_ChCW_LT_LP_Out.Tn_tune	:=	rOpcHC_W[268];
	MM2VIS.tCtr_ChCW_LT_LP_Out.Tv_tune	:=	rOpcHC_W[269];
	MM2VIS.tCtr_ChCW_LT_LP_Out.status	:=	REAL_TO_UINT(rOpcHC_W[270]);
	MM2VIS.tCtr_ChCW_LT_LP_Out.Kp_act	:=	rOpcHC_W[271];
	MM2VIS.tCtr_ChCW_LT_LP_Out.Tn_act	:=	rOpcHC_W[272];
	MM2VIS.tCtr_ChCW_LT_LP_Out.Tv_act	:=	rOpcHC_W[273];

	MM2VIS.rCtr_ChCW_LT_HP_In_X			:=	rOpcHC_W[274];
	MM2VIS.tCtr_ChCW_LT_HP_Out.Y		:=	rOpcHC_W[275];
	MM2VIS.tCtr_ChCW_LT_HP_Out.Y_min_act	:=	rOpcHC_W[276];
	MM2VIS.tCtr_ChCW_LT_HP_Out.Y_max_act	:=	rOpcHC_W[277];
	MM2VIS.tCtr_ChCW_LT_HP_Out.W		:=	rOpcHC_W[278];
	MM2VIS.tCtr_ChCW_LT_HP_Out.e		:=	rOpcHC_W[279];
	MM2VIS.tCtr_ChCW_LT_HP_Out.Kp_tune	:=	rOpcHC_W[280];
	MM2VIS.tCtr_ChCW_LT_HP_Out.Tn_tune	:=	rOpcHC_W[281];
	MM2VIS.tCtr_ChCW_LT_HP_Out.Tv_tune	:=	rOpcHC_W[282];
	MM2VIS.tCtr_ChCW_LT_HP_Out.status	:=	REAL_TO_UINT(rOpcHC_W[283]);
	MM2VIS.tCtr_ChCW_LT_HP_Out.Kp_act	:=	rOpcHC_W[284];
	MM2VIS.tCtr_ChCW_LT_HP_Out.Tn_act	:=	rOpcHC_W[285];
	MM2VIS.tCtr_ChCW_LT_HP_Out.Tv_act	:=	rOpcHC_W[286];

	MM2VIS.rCtr_ECW_In_X		:=	rOpcHC_W[287];
	MM2VIS.tCtr_ECW_Out.Y		:=	rOpcHC_W[288];
	MM2VIS.tCtr_ECW_Out.Y_min_act	:=	rOpcHC_W[289];
	MM2VIS.tCtr_ECW_Out.Y_max_act	:=	rOpcHC_W[290];
	MM2VIS.tCtr_ECW_Out.W		:=	rOpcHC_W[291];
	MM2VIS.tCtr_ECW_Out.e		:=	rOpcHC_W[292];
	MM2VIS.tCtr_ECW_Out.Kp_tune	:=	rOpcHC_W[293];
	MM2VIS.tCtr_ECW_Out.Tn_tune	:=	rOpcHC_W[294];
	MM2VIS.tCtr_ECW_Out.Tv_tune	:=	rOpcHC_W[295];
	MM2VIS.tCtr_ECW_Out.status	:=	REAL_TO_UINT(rOpcHC_W[296]);
	MM2VIS.tCtr_ECW_Out.Kp_act	:=	rOpcHC_W[297];
	MM2VIS.tCtr_ECW_Out.Tn_act	:=	rOpcHC_W[298];
	MM2VIS.tCtr_ECW_Out.Tv_act	:=	rOpcHC_W[299];

	MM2VIS.rCtr_OCW_In_X		:=	rOpcHC_W[300];
	MM2VIS.tCtr_OCW_Out.Y		:=	rOpcHC_W[301];
	MM2VIS.tCtr_OCW_Out.Y_min_act	:=	rOpcHC_W[302];
	MM2VIS.tCtr_OCW_Out.Y_max_act	:=	rOpcHC_W[303];
	MM2VIS.tCtr_OCW_Out.W		:=	rOpcHC_W[304];
	MM2VIS.tCtr_OCW_Out.e		:=	rOpcHC_W[305];
	MM2VIS.tCtr_OCW_Out.Kp_tune	:=	rOpcHC_W[306];
	MM2VIS.tCtr_OCW_Out.Tn_tune	:=	rOpcHC_W[307];
	MM2VIS.tCtr_OCW_Out.Tv_tune	:=	rOpcHC_W[308];
	MM2VIS.tCtr_OCW_Out.status	:=	REAL_TO_UINT(rOpcHC_W[309]);
	MM2VIS.tCtr_OCW_Out.Kp_act	:=	rOpcHC_W[310];
	MM2VIS.tCtr_OCW_Out.Tn_act	:=	rOpcHC_W[311];
	MM2VIS.tCtr_OCW_Out.Tv_act	:=	rOpcHC_W[312];

	MM2VIS.rT_SecCirc_Su			:=	rOpcHC_W[313];
	MM2VIS.rT_BoilerHouse_Su		:=	rOpcHC_W[314];
	MM2VIS.rT_Cooler_ChCW_HT_Re_1_1	:=	rOpcHC_W[315];
	MM2VIS.rT_Cooler_ChCW_HT_Re_1_2	:=	rOpcHC_W[316];
	MM2VIS.rT_Cooler_ChCW_HT_Re_1_3	:=	rOpcHC_W[317];
	MM2VIS.rT_Cooler_ChCW_HT_Re_1_4	:=	rOpcHC_W[318];
	MM2VIS.rT_Cooler_OCW_Re_1_1		:=	rOpcHC_W[319];
	MM2VIS.rT_Cooler_OCW_Re_1_2		:=	rOpcHC_W[320];
	MM2VIS.rT_Cooler_ECW_Re_1_1		:=	rOpcHC_W[321];
	MM2VIS.rT_Cooler_ECW_Re_1_2		:=	rOpcHC_W[322];
	MM2VIS.rT_Cooler_ChCW_LT_Re_1_1	:=	rOpcHC_W[323];
	MM2VIS.rT_Cooler_ChCW_LT_Re_1_2	:=	rOpcHC_W[324];
	MM2VIS.rPr_RW_Su				:=	rOpcHC_W[325];

	MM2VIS.rPr_RW_OCW_Su_2	:=	rOpcHC_W[326];
	MM2VIS.rPosAct_RW_LT_2	:=	rOpcHC_W[327];
	MM2VIS.rPosAct_RW_HT_2	:=	rOpcHC_W[328];
	MM2VIS.rPosAct_RW_ECW_1	:=	rOpcHC_W[329];

	MM2VIS.rPosAct_RW_OCW_1	:=	rOpcHC_W[330];
	MM2VIS.rPosAct_RW_ECW_2	:=	rOpcHC_W[331];
	MM2VIS.rPosAct_RW_OCW_2	:=	rOpcHC_W[332];
	MM2VIS.rT_RW_LT_Re_1	:=	rOpcHC_W[333];
	MM2VIS.rT_RW_LT_Re_2	:=	rOpcHC_W[334];
	MM2VIS.rT_RW_HT_Re_1	:=	rOpcHC_W[335];
	MM2VIS.rT_RW_HT_Re_2	:=	rOpcHC_W[336];
	MM2VIS.rT_RW_ECW_Re_1	:=	rOpcHC_W[337];
	MM2VIS.rT_RW_ECW_Re_2	:=	rOpcHC_W[338];
	MM2VIS.rT_RW_OCW_Re_1	:=	rOpcHC_W[339];

	MM2VIS.rT_RW_OCW_Re_2		:=	rOpcHC_W[340];
	MM2VIS.rSumChC_LT_Stages	:=	rOpcHC_W[341];
	MM2VIS.rSumChC_HT_Stages	:=	rOpcHC_W[342];
	MM2VIS.rSumECW_Stages		:=	rOpcHC_W[343];
	MM2VIS.rSumOCW_Stages		:=	rOpcHC_W[344];

	Para.rECW_Stages_MaxNum		:=	rOpcHC_W[345];
	Para.rOCW_Stages_MaxNum		:=	rOpcHC_W[346];
	Para.rChC_LT_Stages_MaxNum	:=	rOpcHC_W[347];
	Para.rChC_HT_Stages_MaxNum	:=	rOpcHC_W[348];
	Para.iSel_Cooling			:=	REAL_TO_INT(rOpcHC_W[349]);

	MM2VIS.rPr_HR_HT_Su		:=	rOpcHC_W[350];
	MM2VIS.rPr_HR_HT_Re		:=	rOpcHC_W[351];
	MM2VIS.rPr_HR_LT_Su		:=	rOpcHC_W[352];
	MM2VIS.rPr_HR_LT_Re		:=	rOpcHC_W[353];
	MM2VIS.rT_HR_HT_LP_Su	:=	rOpcHC_W[354];
	MM2VIS.rT_HR_HT_LP_Re	:=	rOpcHC_W[355];
	MM2VIS.rT_HR_HT_HP_Su	:=	rOpcHC_W[356];
	MM2VIS.rT_HR_HT_HP_Re	:=	rOpcHC_W[357];
	MM2VIS.rT_HR_LT_LP_Su	:=	rOpcHC_W[358];
	MM2VIS.rT_HR_LT_LP_Re	:=	rOpcHC_W[359];

	MM2VIS.rT_HR_LT_HP_Su	:=	rOpcHC_W[360];
	MM2VIS.rT_HR_LT_HP_Re	:=	rOpcHC_W[361];
    MM2VIS.rT_HR_ECW_Su		:=	rOpcHC_W[362];
	MM2VIS.rT_HR_ECW_Re		:=	rOpcHC_W[363];
	MM2VIS.rT_HR_OCW_Su		:=	rOpcHC_W[364];
	MM2VIS.rT_HR_OCW_Re		:=	rOpcHC_W[365];

	rOpcHC_W[363];
	rOpcHC_W[364];
	rOpcHC_W[365];
	rOpcHC_W[366];
	rOpcHC_W[367];
	rOpcHC_W[368];
	rOpcHC_W[369];

	rOpcHC_W[370];
	rOpcHC_W[371];
	rOpcHC_W[372];
	rOpcHC_W[373];
	rOpcHC_W[374];
	rOpcHC_W[375];
	rOpcHC_W[376];
	rOpcHC_W[377];
	rOpcHC_W[378];
	rOpcHC_W[379];
	rOpcHC_W[380];

	(**BOOL**)
	MM2VIS.tCtr_ChCW_LT_Out.Active			:=	bOpcHC_W[0];
	MM2VIS.tCtr_ChCW_LT_Out.BlockAutoTune	:=	bOpcHC_W[1];
	MM2VIS.tCtr_ChCW_LT_Out.Show_PID_act	:=	bOpcHC_W[2];
	MM2VIS.bLT_HP_Flap_C				:=	bOpcHC_W[3];
	MM2VIS.bLT_HP_Flap_O				:=	bOpcHC_W[4];
	MM2VIS.tCtr_ChCW_HT_Out.Active			:=	bOpcHC_W[5];
	MM2VIS.tCtr_ChCW_HT_Out.BlockAutoTune	:=	bOpcHC_W[6];
	MM2VIS.tCtr_ChCW_HT_Out.Show_PID_act	:=	bOpcHC_W[7];
	MM2VIS.bLT_LP_Flap_C				:=	bOpcHC_W[8];
	MM2VIS.bLT_LP_Flap_O				:=	bOpcHC_W[9];

	MM2VIS.tCtr_ChCW_HT_LP_Out.Active			:=	bOpcHC_W[10];
	MM2VIS.tCtr_ChCW_HT_LP_Out.BlockAutoTune	:=	bOpcHC_W[11];
	MM2VIS.tCtr_ChCW_HT_LP_Out.Show_PID_act		:=	bOpcHC_W[12];
	MM2VIS.bDem_LT_HP_PreHeat				:=	bOpcHC_W[13];
	MM2VIS.bDem_LT_LP_PreHeat				:=	bOpcHC_W[14];
	MM2VIS.tCtr_ChCW_HT_HP_Out.Active			:=	bOpcHC_W[15];
	MM2VIS.tCtr_ChCW_HT_HP_Out.BlockAutoTune	:=	bOpcHC_W[16];
	MM2VIS.tCtr_ChCW_HT_HP_Out.Show_PID_act		:=	bOpcHC_W[17];
	MM2VIS.bDem_HR_CircPump_HT_1		:=	bOpcHC_W[18];
	MM2VIS.bDem_HR_CircPump_HT_2		:=	bOpcHC_W[19];

	MM2VIS.tCtr_ChCW_LT_LP_Out.Active			:=	bOpcHC_W[20];
	MM2VIS.tCtr_ChCW_LT_LP_Out.BlockAutoTune	:=	bOpcHC_W[21];
	MM2VIS.tCtr_ChCW_LT_LP_Out.Show_PID_act		:=	bOpcHC_W[22];
	MM2VIS.bDem_HR_CircPump_LT_1		:=	bOpcHC_W[23];
	MM2VIS.bDem_HR_CircPump_LT_2		:=	bOpcHC_W[24];
	MM2VIS.tCtr_ChCW_LT_HP_Out.Active			:=	bOpcHC_W[25];
	MM2VIS.tCtr_ChCW_LT_HP_Out.BlockAutoTune	:=	bOpcHC_W[26];
	MM2VIS.tCtr_ChCW_LT_HP_Out.Show_PID_act		:=	bOpcHC_W[27];
	MM2VIS.bDem_HR_CircPump_ECW_1		:=	bOpcHC_W[28];
	MM2VIS.bDem_HR_CircPump_ECW_2		:=	bOpcHC_W[29];

	MM2VIS.tCtr_ECW_Out.Active			:=	bOpcHC_W[30];
	MM2VIS.tCtr_ECW_Out.BlockAutoTune	:=	bOpcHC_W[31];
	MM2VIS.tCtr_ECW_Out.Show_PID_act	:=	bOpcHC_W[32];
	MM2VIS.bDem_HR_CircPump_OCW_1		:=	bOpcHC_W[33];
	MM2VIS.bDem_HR_CircPump_OCW_2		:=	bOpcHC_W[34];
	MM2VIS.tCtr_OCW_Out.Active			:=	bOpcHC_W[35];
	MM2VIS.tCtr_OCW_Out.BlockAutoTune	:=	bOpcHC_W[36];
	MM2VIS.tCtr_OCW_Out.Show_PID_act	:=	bOpcHC_W[37];
	bOpcHC_W[38];
	bOpcHC_W[39];

	bOpcHC_W[40];
	bOpcHC_W[41];
	bOpcHC_W[42];
	bOpcHC_W[43];
	bOpcHC_W[44];

	MM2VIS.bDem_Cooler_ChCW_LT_1	:=	bOpcHC_W[45];
	MM2VIS.bDem_Cooler_ChCW_LT_2	:=	bOpcHC_W[46];
	MM2VIS.bDem_Cooler_ChCW_HT_1	:=	bOpcHC_W[47];
	MM2VIS.bDem_Cooler_ChCW_HT_2	:=	bOpcHC_W[48];
	bPreHeatWDayLT_On				:=	bOpcHC_W[49];

	MM2VIS.bDem_Cooler_ChCW_LT_LP_2	:=	bOpcHC_W[50];
	MM2VIS.bDem_Cooler_ChCW_LT_HP_1	:=	bOpcHC_W[51];
	MM2VIS.bDem_Cooler_ChCW_LT_HP_2	:=	bOpcHC_W[52];
	MM2VIS.bDem_Cooler_ChCW_HT_LP_1	:=	bOpcHC_W[53];
	MM2VIS.bDem_Cooler_ChCW_HT_LP_2	:=	bOpcHC_W[54];
	MM2VIS.bDem_Cooler_ChCW_HT_HP_1	:=	bOpcHC_W[55];
	MM2VIS.bDem_Cooler_ChCW_HT_HP_2	:=	bOpcHC_W[56];
	MM2VIS.bDem_Cooler_ECW_1		:=	bOpcHC_W[57];
	MM2VIS.bDem_Cooler_ECW_2		:=	bOpcHC_W[58];
	MM2VIS.bDem_Cooler_OCW_1		:=	bOpcHC_W[59];

	MM2VIS.bDem_Cooler_OCW_2		:=	bOpcHC_W[60];
	MM2VIS.bDem_ChCW_LT_Pump		:=	bOpcHC_W[61];
	MM2VIS.bDem_ChCW_HT_Pump		:=	bOpcHC_W[62];
	MM2VIS.bDem_ChCW_LT_LP_Pump		:=	bOpcHC_W[63];
	MM2VIS.bDem_ChCW_LT_HP_Pump		:=	bOpcHC_W[64];
	MM2VIS.bDem_ChCW_HT_LP_Pump		:=	bOpcHC_W[65];
	MM2VIS.bDem_ChCW_HT_HP_Pump		:=	bOpcHC_W[66];
	MM2VIS.bDem_ECW_Pump			:=	bOpcHC_W[67];
	MM2VIS.bDem_OCW_Pump			:=	bOpcHC_W[68];
	MM2VIS.bPs_ChCW_LT_bEngine_Hi	:=	bOpcHC_W[69];

	MM2VIS.bPs_ChCW_HT_bEngine_Hi		:=	bOpcHC_W[70];
	MM2VIS.bPs_ChCW_LT_LP_bEngine_Hi	:=	bOpcHC_W[71];
	MM2VIS.bPs_ChCW_LT_HP_bEngine_Hi	:=	bOpcHC_W[72];
	MM2VIS.bPs_ChCW_HT_LP_bEngine_Hi	:=	bOpcHC_W[73];
	MM2VIS.bPs_ChCW_HT_HP_bEngine_Hi	:=	bOpcHC_W[74];
	MM2VIS.bPs_ECW_bEngine_Hi			:=	bOpcHC_W[75];
	MM2VIS.bPs_OCW_bEngine_Hi			:=	bOpcHC_W[76];
	MM2VIS.bPs_ChCW_LT_bPump_Low		:=	bOpcHC_W[77];
	MM2VIS.bPs_ChCW_HT_bPump_Low		:=	bOpcHC_W[78];
	MM2VIS.bPs_ChCW_LT_LP_bPump_Low		:=	bOpcHC_W[79];

	MM2VIS.bPs_ChCW_LT_HP_bPump_Low		:=	bOpcHC_W[80];
	MM2VIS.bPs_ChCW_HT_LP_bPump_Low		:=	bOpcHC_W[81];
	MM2VIS.bPs_ChCW_HT_HP_bPump_Low		:=	bOpcHC_W[82];
	MM2VIS.bPs_ECW_bPump_Low			:=	bOpcHC_W[83];
	MM2VIS.bPs_OCW_bPump_Low			:=	bOpcHC_W[84];
	MM2VIS.bTs_ChCW_LT_bEngine_Hi		:=	bOpcHC_W[85];
	MM2VIS.bTs_ChCW_HT_bEngine_Hi		:=	bOpcHC_W[86];
	MM2VIS.bTs_ChCW_LT_LP_bEngine_Hi	:=	bOpcHC_W[87];
	MM2VIS.bTs_ChCW_LT_HP_bEngine_Hi	:=	bOpcHC_W[88];
	MM2VIS.bTs_ChCW_HT_LP_bEngine_Hi	:=	bOpcHC_W[89];

	MM2VIS.bTs_ChCW_HT_HP_bEngine_Hi	:=	bOpcHC_W[90];
	MM2VIS.bTs_ECW_bEngine_Hi			:=	bOpcHC_W[91];
	MM2VIS.bTs_OCW_bEngine_Hi			:=	bOpcHC_W[92];
	MM2VIS.bCooler_ChCW_LT_1_Op			:=	bOpcHC_W[93];
	MM2VIS.bCooler_ChCW_LT_2_Op			:=	bOpcHC_W[94];
	MM2VIS.bCooler_ChCW_HT_1_Op			:=	bOpcHC_W[95];
	MM2VIS.bCooler_ChCW_HT_2_Op			:=	bOpcHC_W[96];
	MM2VIS.bCooler_ChCW_LT_LP_1_Op		:=	bOpcHC_W[97];
	MM2VIS.bCooler_ChCW_LT_LP_2_Op		:=	bOpcHC_W[98];
	MM2VIS.bCooler_ChCW_LT_HP_1_Op		:=	bOpcHC_W[99];

	MM2VIS.bCooler_ChCW_LT_HP_2_Op	:=	bOpcHC_W[100];
	MM2VIS.bCooler_ChCW_HT_LP_1_Op	:=	bOpcHC_W[101];
	MM2VIS.bCooler_ChCW_HT_LP_2_Op	:=	bOpcHC_W[102];
	MM2VIS.bCooler_ChCW_HT_HP_1_Op	:=	bOpcHC_W[103];
	MM2VIS.bCooler_ChCW_HT_HP_2_Op	:=	bOpcHC_W[104];
	MM2VIS.bCooler_ECW_1_Op			:=	bOpcHC_W[105];
	MM2VIS.bCooler_ECW_2_Op			:=	bOpcHC_W[106];
	MM2VIS.bCooler_OCW_1_Op			:=	bOpcHC_W[107];
	MM2VIS.bCooler_OCW_2_Op			:=	bOpcHC_W[108];
	MM2VIS.bPs_RW_Low				:=	bOpcHC_W[109];

	MM2VIS.bTs_RW_Hi				:=	bOpcHC_W[110];
	MM2VIS.bPs_ChCW_LT_aEngine_Low	:=	bOpcHC_W[111];
	MM2VIS.bPs_ChCW_HT_aEngine_Low	:=	bOpcHC_W[112];
	MM2VIS.bPs_ChCW_LT_LP_aEngine_Low	:=	bOpcHC_W[113];
	MM2VIS.bPs_ChCW_LT_HP_aEngine_Low	:=	bOpcHC_W[114];
	MM2VIS.bPs_ChCW_HT_LP_aEngine_Low	:=	bOpcHC_W[115];
	MM2VIS.bPs_ChCW_HT_HP_aEngine_Low	:=	bOpcHC_W[116];
	MM2VIS.bPs_ECW_aEngine_Low		:=	bOpcHC_W[117];
	MM2VIS.bPs_OCW_aEngine_Low		:=	bOpcHC_W[118];
	MM2VIS.bFlow_BoilerHouse_Lo		:=	bOpcHC_W[119];

	MM2VIS.bPs_BoilerHouse_Hi		:=	bOpcHC_W[120];
	MM2VIS.bPs_BoilerHouse_Lo		:=	bOpcHC_W[121];
	MM2VIS.bTs_BoilerHouse_Hi		:=	bOpcHC_W[122];
	MM2VIS.bFlow_SecCirc_Lo			:=	bOpcHC_W[123];
	MM2VIS.bPs_SecCirc_Hi			:=	bOpcHC_W[124];
	MM2VIS.bPs_SecCirc_Lo			:=	bOpcHC_W[125];
	MM2VIS.bTs_SecCirc_Hi			:=	bOpcHC_W[126];
	MM2VIS.bDem_BoilerHouse_Pump	:=	bOpcHC_W[127];
	MM2VIS.bDem_SecCirc_Pump		:=	bOpcHC_W[128];
	bOpcHC_W[129];
	bOpcHC_W[130];

	(*Parameter für Vis*)
	Para.bPs_bPumpLowActive			:= bOpcHC_W[131];
	Para.bPs_bEngineHiActive		:= bOpcHC_W[132];
	Para.bTs_bEngineHiActive		:= bOpcHC_W[133];
	Para.bPs_aEngineLowActive		:= bOpcHC_W[134];
	Para.bT_bCV_Active				:= bOpcHC_W[135];
	Para.bFB_CC_Active				:= bOpcHC_W[136];
	Para.bFB_Cooler_Active			:= bOpcHC_W[137];
	Para.bT_Cooler_Re_Active		:= bOpcHC_W[138];
	Para.bPr_Cooler_Re_Active		:= bOpcHC_W[139];
	Para.bT_Cooler_Su_Active		:= bOpcHC_W[140];
	Para.bPr_Cooler_Su_Active		:= bOpcHC_W[141];
	Para.bT_RW_Re_Active			:= bOpcHC_W[142];
	Para.bT_RW_Su_Active			:= bOpcHC_W[143];
	Para.bTs_RW_Active				:= bOpcHC_W[144];
	Para.bPs_RW_Active				:= bOpcHC_W[145];
	Para.bCtr_ECW					:= bOpcHC_W[146];
	Para.bCtr_OCW					:= bOpcHC_W[147];
	Para.bCtr_ChCW_LT				:= bOpcHC_W[148];
	Para.bCtr_ChCW_LT_LP			:= bOpcHC_W[149];
	Para.bCtr_ChCW_LT_HP			:= bOpcHC_W[150];
	Para.bCtr_ChCW_HT				:= bOpcHC_W[151];
	Para.bCtr_ChCW_HT_LP			:= bOpcHC_W[152];
	Para.bCtr_ChCW_HT_HP			:= bOpcHC_W[153];

	Para.bDem_Cooler_ECW_1			:= bOpcHC_W[154];
	Para.bDem_Cooler_ECW_2			:= bOpcHC_W[155];
	Para.bVol_ECW_Re				:= bOpcHC_W[156];
	Para.bVol_ECW_Su				:= bOpcHC_W[157];
	Para.bT_ECW_Re					:= bOpcHC_W[158];
	Para.bPr_ECW_Re					:= bOpcHC_W[159];
	Para.bT_ECW_IC_Re				:= bOpcHC_W[160];
	Para.bPr_ECW_IC_Re				:= bOpcHC_W[161];
	Para.bT_ECW_Su					:= bOpcHC_W[162];
	Para.bPr_ECW_Su					:= bOpcHC_W[163];
	Para.bT_ECW_IC_Su				:= bOpcHC_W[164];
	Para.bPr_ECW_IC_Su				:= bOpcHC_W[165];
	Para.bECW_Stages_Active			:= bOpcHC_W[166];

	Para.bDem_Cooler_OCW_1			:= bOpcHC_W[167];
	Para.bDem_Cooler_OCW_2			:= bOpcHC_W[168];
	Para.bVol_OCW_Re				:= bOpcHC_W[169];
	Para.bVol_OCW_Su				:= bOpcHC_W[170];
	Para.bT_OCW_Re					:= bOpcHC_W[171];
	Para.bPr_OCW_Re					:= bOpcHC_W[172];
	Para.bT_OCW_IC_Re				:= bOpcHC_W[173];
	Para.bPr_OCW_IC_Re				:= bOpcHC_W[174];
	Para.bT_OCW_Su					:= bOpcHC_W[175];
	Para.bPr_OCW_Su					:= bOpcHC_W[176];
	Para.bT_OCW_IC_Su				:= bOpcHC_W[177];
	Para.bPr_OCW_IC_Su				:= bOpcHC_W[178];
	Para.bOCW_Stages_Active			:= bOpcHC_W[179];

	Para.bDem_Cooler_ChCW_LT_1		:= bOpcHC_W[180];
	Para.bDem_Cooler_ChCW_LT_2		:= bOpcHC_W[181];
	Para.bVol_ChCW_Re_LT			:= bOpcHC_W[182];
	Para.bVol_ChCW_Su_LT			:= bOpcHC_W[183];
	Para.bT_ChCW_Re_LT				:= bOpcHC_W[184];
	Para.bPr_ChCW_Re_LT				:= bOpcHC_W[185];
	Para.bT_ChCW_LT_IC_Re			:= bOpcHC_W[186];
	Para.bPr_ChCW_LT_IC_Re			:= bOpcHC_W[187];
	Para.bT_ChCW_Su_LT				:= bOpcHC_W[188];
	Para.bPr_ChCW_Su_LT				:= bOpcHC_W[189];
	Para.bT_ChCW_LT_IC_Su			:= bOpcHC_W[190];
	Para.bPr_ChCW_LT_IC_Su			:= bOpcHC_W[191];
	Para.bChC_LT_Stages_Active		:= bOpcHC_W[192];

	Para.bDem_Cooler_ChCW_HT_1		:= bOpcHC_W[193];
	Para.bDem_Cooler_ChCW_HT_2		:= bOpcHC_W[194];
	Para.bVol_ChCW_Re_HT			:= bOpcHC_W[195];
	Para.bVol_ChCW_Su_HT			:= bOpcHC_W[196];
	Para.bT_ChCW_Re_HT				:= bOpcHC_W[197];
	Para.bPr_ChCW_Re_HT				:= bOpcHC_W[198];
	Para.bT_ChCW_HT_IC_Re			:= bOpcHC_W[199];
	Para.bPr_ChCW_HT_IC_Re			:= bOpcHC_W[200];
	Para.bT_ChCW_Su_HT				:= bOpcHC_W[201];
	Para.bPr_ChCW_Su_HT				:= bOpcHC_W[202];
	Para.bT_ChCW_HT_IC_Su			:= bOpcHC_W[203];
	Para.bPr_ChCW_HT_IC_Su			:= bOpcHC_W[204];
	Para.bChC_HT_Stages_Active		:= bOpcHC_W[205];

	Para.bDem_Cooler_ChCW_LT_LP_1	:= bOpcHC_W[206];
	Para.bDem_Cooler_ChCW_LT_LP_2	:= bOpcHC_W[207];
	Para.bVol_ChCW_Re_LT_LP			:= bOpcHC_W[208];
	Para.bVol_ChCW_Su_LT_LP			:= bOpcHC_W[209];
	Para.bT_ChCW_Re_LT_LP			:= bOpcHC_W[210];
	Para.bPr_ChCW_Re_LT_LP			:= bOpcHC_W[211];
	Para.bT_ChCW_LT_LP_IC_Re		:= bOpcHC_W[212];
	Para.bPr_ChCW_LT_LP_IC_Re		:= bOpcHC_W[213];
	Para.bT_ChCW_Su_LT_LP			:= bOpcHC_W[214];
	Para.bPr_ChCW_Su_LT_LP			:= bOpcHC_W[215];
	Para.bT_ChCW_LT_LP_IC_Su		:= bOpcHC_W[216];
	Para.bPr_ChCW_LT_LP_IC_Su		:= bOpcHC_W[217];

	Para.bDem_Cooler_ChCW_LT_HP_1	:= bOpcHC_W[218];
	Para.bDem_Cooler_ChCW_LT_HP_2	:= bOpcHC_W[219];
	Para.bVol_ChCW_Re_LT_HP			:= bOpcHC_W[220];
	Para.bVol_ChCW_Su_LT_HP			:= bOpcHC_W[221];
	Para.bT_ChCW_Re_LT_HP			:= bOpcHC_W[222];
	Para.bPr_ChCW_Re_LT_HP			:= bOpcHC_W[223];
	Para.bT_ChCW_LT_HP_IC_Re		:= bOpcHC_W[224];
	Para.bPr_ChCW_LT_HP_IC_Re		:= bOpcHC_W[225];
	Para.bT_ChCW_Su_LT_HP			:= bOpcHC_W[226];
	Para.bPr_ChCW_Su_LT_HP			:= bOpcHC_W[227];
	Para.bT_ChCW_LT_HP_IC_Su		:= bOpcHC_W[228];
	Para.bPr_ChCW_LT_HP_IC_Su		:= bOpcHC_W[229];

	Para.bDem_Cooler_ChCW_HT_LP_1	:= bOpcHC_W[230];
	Para.bDem_Cooler_ChCW_HT_LP_2	:= bOpcHC_W[231];
	Para.bVol_ChCW_Re_HT_LP			:= bOpcHC_W[232];
	Para.bVol_ChCW_Su_HT_LP			:= bOpcHC_W[233];
	Para.bT_ChCW_Re_HT_LP			:= bOpcHC_W[234];
	Para.bPr_ChCW_Re_HT_LP			:= bOpcHC_W[235];
	Para.bT_ChCW_HT_LP_IC_Re		:= bOpcHC_W[236];
	Para.bPr_ChCW_HT_LP_IC_Re		:= bOpcHC_W[237];
	Para.bT_ChCW_Su_HT_LP			:= bOpcHC_W[238];
	Para.bPr_ChCW_Su_HT_LP			:= bOpcHC_W[239];
	Para.bT_ChCW_HT_LP_IC_Su		:= bOpcHC_W[240];
	Para.bPr_ChCW_HT_LP_IC_Su		:= bOpcHC_W[241];

	Para.bDem_Cooler_ChCW_HT_HP_1	:= bOpcHC_W[242];
	Para.bDem_Cooler_ChCW_HT_HP_2	:= bOpcHC_W[243];
	Para.bVol_ChCW_Re_HT_HP			:= bOpcHC_W[244];
	Para.bVol_ChCW_Su_HT_HP			:= bOpcHC_W[245];
	Para.bT_ChCW_Re_HT_HP			:= bOpcHC_W[246];
	Para.bPr_ChCW_Re_HT_HP			:= bOpcHC_W[247];
	Para.bT_ChCW_HT_HP_IC_Re		:= bOpcHC_W[248];
	Para.bPr_ChCW_HT_HP_IC_Re		:= bOpcHC_W[249];
	Para.bT_ChCW_Su_HT_HP			:= bOpcHC_W[250];
	Para.bPr_ChCW_Su_HT_HP			:= bOpcHC_W[251];
	Para.bT_ChCW_HT_HP_IC_Su		:= bOpcHC_W[252];
	Para.bPr_ChCW_HT_HP_IC_Su		:= bOpcHC_W[253];

	MM2VIS.bDem_Cooler_X				:=	bOpcHC_W[254];

END_PROGRAM
```

### Program Logical/DataInterface/OpcME (IEC) - OPC Var for Testbench

#### OpcME.st
```iecst
(*******************************************************************************
OpcME	 Variables read or write to Testbench

This code is confidential AND proprietary to the INNIO Company.
It may NOT be used in any form, or reproduced in any manner, without the express
written permission of the INNIO Company.
Copyright, INNIO Company, 2022

- list addidtional customized IO channels

Customized modifications: -
------------------------

History:
-------
V1.00.0	14.09.2022	Vockenberger	Neu erstellt
V1.01.0	23.07.2023	Vockenberger	Ext Vorgaben von MDE eingefügt
		28.07.2023	Vockenberger	Struktur von OPC_DI geändert
V1.03.0 10.06.2025	Vockenberger	added extern setpoint for CAT temp over MDE

Instructions FOR use:
--------------------

Outstandings:
------------

*******************************************************************************)

PROGRAM _CYCLIC

	(**Wird von Motor-CPU geschrieben**********************)
	(**REAL**)
	rOpcME_R[0] :=	IN_DI.rCAT_TempSet;
	rOpcME_R[1];
	rOpcME_R[2];
	rOpcME_R[3];
	rOpcME_R[4];
	rOpcME_R[5];
	rOpcME_R[6];
	rOpcME_R[7];
	rOpcME_R[8];
	rOpcME_R[9];
	rOpcME_R[10];

	(**BOOL**)
	bOpcME_R[0]	:=	VIS2MM.bExtLeanox_ActiveMDE;
	bOpcME_R[1]	:=	VIS2MM.bCA_IgnP_ActiveMDE;
	bOpcME_R[2]	:=	VIS2MM.bExtMN_ActiveMDE;
	bOpcME_R[3] :=	VIS2MM.bExtNOX_ActiveMDE;
	bOpcME_R[4] :=	VIS2MM.bExtCAT_TempActive;
	bOpcME_R[5];
	bOpcME_R[6];
	bOpcME_R[7];
	bOpcME_R[8];
	bOpcME_R[9];
	bOpcME_R[10];

	(*Measurement from Testbench*)
	rP_MDE_OPC_Set					:= rOpcME_W[0];
	MM2VIS.rStartpointCA_IgnP_Set 	:= rOpcME_W[1];
	MM2VIS.rStartpointLamEngLL_Set 	:= rOpcME_W[2];
	MM2VIS.rStartpoint_p2_Set 		:= rOpcME_W[3];
	MM2VIS.rExtMN_Set 				:= rOpcME_W[4];
	MM2VIS.rLam_Eng_LL_ManSet_Cust 	:= rOpcME_W[5];
	MM2VIS.rPr_Leanox_ManSet_Cust 	:= rOpcME_W[6];
	MM2VIS.rCA_IgnP_CylOffset[1] 	:= rOpcME_W[7];
	MM2VIS.rCA_IgnP_CylOffset[2] 	:= rOpcME_W[8];
	MM2VIS.rCA_IgnP_CylOffset[3] 	:= rOpcME_W[9];

	MM2VIS.rCA_IgnP_CylOffset[4] 	:= rOpcME_W[10];
	MM2VIS.rCA_IgnP_CylOffset[5] 	:= rOpcME_W[11];
	MM2VIS.rCA_IgnP_CylOffset[6] 	:= rOpcME_W[12];
	MM2VIS.rCA_IgnP_CylOffset[7] 	:= rOpcME_W[13];
	MM2VIS.rCA_IgnP_CylOffset[8] 	:= rOpcME_W[14];
	MM2VIS.rCA_IgnP_CylOffset[9] 	:= rOpcME_W[15];
	MM2VIS.rCA_IgnP_CylOffset[10] 	:= rOpcME_W[16];
	MM2VIS.rCA_IgnP_CylOffset[11] 	:= rOpcME_W[17];
	MM2VIS.rCA_IgnP_CylOffset[12] 	:= rOpcME_W[18];
	MM2VIS.rCA_IgnP_CylOffset[13] 	:= rOpcME_W[19];

	MM2VIS.rCA_IgnP_CylOffset[14] 	:= rOpcME_W[20];
	MM2VIS.rCA_IgnP_CylOffset[15] 	:= rOpcME_W[21];
	MM2VIS.rCA_IgnP_CylOffset[16] 	:= rOpcME_W[22];
	MM2VIS.rCA_IgnP_CylOffset[17] 	:= rOpcME_W[23];
	MM2VIS.rCA_IgnP_CylOffset[18] 	:= rOpcME_W[24];
	MM2VIS.rCA_IgnP_CylOffset[19] 	:= rOpcME_W[25];
	MM2VIS.rCA_IgnP_CylOffset[20] 	:= rOpcME_W[26];
	MM2VIS.rCA_IgnP_CylOffset[21] 	:= rOpcME_W[27];
	MM2VIS.rCA_IgnP_CylOffset[22] 	:= rOpcME_W[28];
	MM2VIS.rCA_IgnP_CylOffset[23] 	:= rOpcME_W[29];

	MM2VIS.rCA_IgnP_CylOffset[24] 	:= rOpcME_W[30];
	MM2VIS.rStartpoint_MN_Set	  	:= rOpcME_W[31];
	MM2VIS.rCA_IgnPFromMDE	 	  	:= rOpcME_W[32];
	MM2VIS.rNOX_ManSet_Cust			:= rOpcME_W[33];
	MM2VIS.rStartpoint_NOX_Set		:= rOpcME_W[34];
	MM2VIS.rNOX_FromMDE				:= rOpcME_W[35];
	MM2VIS.rStatusExhaustMde		:= rOpcME_W[36];
	MM2VIS.rExtCAT_TempSetMDE		:= rOpcME_W[37];
	OUT_DI.rExtCAT_TempSet			:= rOpcME_W[38];
	MM2VIS.rStartpoint_CAT_Temp_Set	:= rOpcME_W[39];

	rOpcME_W[40];
	rOpcME_W[41];
	rOpcME_W[42];
	rOpcME_W[43];
	rOpcME_W[44];
	rOpcME_W[45];
	rOpcME_W[46];
	rOpcME_W[47];
	rOpcME_W[48];
	rOpcME_W[49];
	rOpcME_W[50];

	(**BOOL**)
	bMDEBusAlive 				:= bOpcME_W[0];
	bMDEOPC_Dem 				:= bOpcME_W[1];
	MM2VIS.bLeanox_Man_Cust 	:= bOpcME_W[2];
	MM2VIS.bCA_IgnP_CylOffset_Active := bOpcME_W[3];
	MM2VIS.bExtMN_Active 	 	:= bOpcME_W[4];
	MM2VIS.bExtLeanoxFromMDE 	:= bOpcME_W[5];
	MM2VIS.bCA_IgnPFromMDE 	 	:= bOpcME_W[6];
	MM2VIS.bExtMNFromMDE 	 	:= bOpcME_W[7];
	MM2VIS.bExtNOXFromMDE	 	:= bOpcME_W[8];
	MM2VIS.bExtNOX_Active	 	:= bOpcME_W[9];
	MM2VIS.bExtCAT_TempActiveMDE:= bOpcME_W[10];

	OUT_DI.bExtCAT_Temp_Active	:= bOpcME_W[11];
	bOpcME_W[12];
	bOpcME_W[13];
	bOpcME_W[14];
	bOpcME_W[15];
	bOpcME_W[16];
	bOpcME_W[17];
	bOpcME_W[18];
	bOpcME_W[19];
	bOpcME_W[20];

END_PROGRAM
```

### Program Logical/DataInterface/OpcMsg (IEC) - OPC Var for Testbench

#### OpcMsg.st
```iecst
(*******************************************************************************
OpcMsg	 Variables read from Testbench

This code is confidential AND proprietary to the INNIO Company.
It may NOT be used in any form, or reproduced in any manner, without the express
written permission of the INNIO Company.
Copyright, INNIO Company, 2022

- list addidtional customized IO channels

Customized modifications: -
------------------------

History:
-------
V1.00.0	14.09.2022		Vockenberger	Neu erstellt
V1.01.0	20.07.2023		Vockenberger	Neue Störungen/Warnungen eingefügt
		28.07.2023		Vockenberger	Struktur von OPC_DI geändert
V1.01.1	18.03.2024		Gruber St.		added messages bMsg7625 to bMsg7650
V1.02.0	20.03.2024		Vockenberger	Heizhaus, V-Kühler und Transformator Störungen hinzugefügt

Instructions FOR use:
--------------------

Outstandings:
------------

*******************************************************************************)

PROGRAM _CYCLIC

	(**BOOL**)
	TON_bComOpcBitTB(IN:= bComOpcBitTB, PT:=T#1s);
	IF TON_bComOpcBitTB.Q THEN
		bOpcMsg_W[0] := FALSE;
	END_IF
	TON_bComOpcFailTB(IN:= NOT bOpcMsg_W[0], PT:=T#1s);
	IF TON_bComOpcFailTB.Q OR TON_bComOpcFailMDE.Q THEN
		MM2VIS.bMsg7000 := TRUE;
	ELSE
		MM2VIS.bMsg7000 := FALSE;
	END_IF
	bComOpcBitTB	:=	bOpcMsg_W[0];
	MM2VIS.bMsg7001	:=	bOpcMsg_W[1];
	MM2VIS.bMsg7002	:=	bOpcMsg_W[2];
	MM2VIS.bMsg7003	:=	bOpcMsg_W[3];
	MM2VIS.bMsg7004	:=	bOpcMsg_W[4];
	MM2VIS.bMsg7005	:=	bOpcMsg_W[5];
	MM2VIS.bMsg7006	:=	bOpcMsg_W[6];
	MM2VIS.bMsg7007	:=	bOpcMsg_W[7];
	MM2VIS.bMsg7008	:=	bOpcMsg_W[8];
	MM2VIS.bMsg7009	:=	bOpcMsg_W[9];
	MM2VIS.bMsg7010	:=	bOpcMsg_W[10];
	MM2VIS.bMsg7011	:=	bOpcMsg_W[11];
	MM2VIS.bMsg7012	:=	bOpcMsg_W[12];
	MM2VIS.bMsg7013	:=	bOpcMsg_W[13];
	MM2VIS.bMsg7014	:=	bOpcMsg_W[14];
	MM2VIS.bMsg7015	:=	bOpcMsg_W[15];
	MM2VIS.bMsg7016	:=	bOpcMsg_W[16];
	MM2VIS.bMsg7017	:=	bOpcMsg_W[17];
	MM2VIS.bMsg7018	:=	bOpcMsg_W[18];
	MM2VIS.bMsg7019	:=	bOpcMsg_W[19];
	MM2VIS.bMsg7020	:=	bOpcMsg_W[20];
	MM2VIS.bMsg7021	:=	bOpcMsg_W[21];
	MM2VIS.bMsg7022	:=	bOpcMsg_W[22];
	MM2VIS.bMsg7023	:=	bOpcMsg_W[23];
	MM2VIS.bMsg7024	:=	bOpcMsg_W[24];
	MM2VIS.bMsg7025	:=	bOpcMsg_W[25];
	MM2VIS.bMsg7026	:=	bOpcMsg_W[26];
	MM2VIS.bMsg7027	:=	bOpcMsg_W[27];
	MM2VIS.bMsg7028	:=	bOpcMsg_W[28];
	MM2VIS.bMsg7029	:=	bOpcMsg_W[29];
	MM2VIS.bMsg7030	:=	bOpcMsg_W[30];
	MM2VIS.bMsg7031	:=	bOpcMsg_W[31];
	MM2VIS.bMsg7032	:=	bOpcMsg_W[32];
	MM2VIS.bMsg7033	:=	bOpcMsg_W[33];
	MM2VIS.bMsg7034	:=	bOpcMsg_W[34];
	MM2VIS.bMsg7035	:=	bOpcMsg_W[35];
	MM2VIS.bMsg7036	:=	bOpcMsg_W[36];
	MM2VIS.bMsg7037	:=	bOpcMsg_W[37];
	MM2VIS.bMsg7038	:=	bOpcMsg_W[38];
	MM2VIS.bMsg7039	:=	bOpcMsg_W[39];
	MM2VIS.bMsg7040	:=	bOpcMsg_W[40];
	MM2VIS.bMsg7041	:=	bOpcMsg_W[41];
	MM2VIS.bMsg7042	:=	bOpcMsg_W[42];
	MM2VIS.bMsg7043	:=	bOpcMsg_W[43];
	MM2VIS.bMsg7044	:=	bOpcMsg_W[44];
	MM2VIS.bMsg7045	:=	bOpcMsg_W[45];
	MM2VIS.bMsg7046	:=	bOpcMsg_W[46];
	MM2VIS.bMsg7047	:=	bOpcMsg_W[47];
	MM2VIS.bMsg7048	:=	bOpcMsg_W[48];
	MM2VIS.bMsg7049	:=	bOpcMsg_W[49];
	MM2VIS.bMsg7050	:=	bOpcMsg_W[50];
	MM2VIS.bMsg7051	:=	bOpcMsg_W[51];
	MM2VIS.bMsg7052	:=	bOpcMsg_W[52];
	MM2VIS.bMsg7053	:=	bOpcMsg_W[53];
	MM2VIS.bMsg7054	:=	bOpcMsg_W[54];
	MM2VIS.bMsg7055	:=	bOpcMsg_W[55];
	MM2VIS.bMsg7056	:=	bOpcMsg_W[56];
	MM2VIS.bMsg7057	:=	bOpcMsg_W[57];
	MM2VIS.bMsg7058	:=	bOpcMsg_W[58];
	MM2VIS.bMsg7059	:=	bOpcMsg_W[59];
	MM2VIS.bMsg7060	:=	bOpcMsg_W[60];
	MM2VIS.bMsg7061	:=	bOpcMsg_W[61];
	MM2VIS.bMsg7062	:=	bOpcMsg_W[62];
	MM2VIS.bMsg7063	:=	bOpcMsg_W[63];
	MM2VIS.bMsg7064	:=	bOpcMsg_W[64];
	MM2VIS.bMsg7065	:=	bOpcMsg_W[65];
	MM2VIS.bMsg7066	:=	bOpcMsg_W[66];
	MM2VIS.bMsg7067	:=	bOpcMsg_W[67];
	MM2VIS.bMsg7068	:=	bOpcMsg_W[68];
	MM2VIS.bMsg7069	:=	bOpcMsg_W[69];
	MM2VIS.bMsg7070	:=	bOpcMsg_W[70];
	MM2VIS.bMsg7071	:=	bOpcMsg_W[71];
	MM2VIS.bMsg7072	:=	bOpcMsg_W[72];
	MM2VIS.bMsg7073	:=	bOpcMsg_W[73];
	MM2VIS.bMsg7074	:=	bOpcMsg_W[74];
	MM2VIS.bMsg7075	:=	bOpcMsg_W[75];
	MM2VIS.bMsg7076	:=	bOpcMsg_W[76];
	MM2VIS.bMsg7077	:=	bOpcMsg_W[77];
	MM2VIS.bMsg7078	:=	bOpcMsg_W[78];
	MM2VIS.bMsg7079	:=	bOpcMsg_W[79];
	MM2VIS.bMsg7080	:=	bOpcMsg_W[80];
	MM2VIS.bMsg7081	:=	bOpcMsg_W[81];
	MM2VIS.bMsg7082	:=	bOpcMsg_W[82];
	MM2VIS.bMsg7083	:=	bOpcMsg_W[83];
	MM2VIS.bMsg7084	:=	bOpcMsg_W[84];
	MM2VIS.bMsg7085	:=	bOpcMsg_W[85];
	MM2VIS.bMsg7086	:=	bOpcMsg_W[86];
	MM2VIS.bMsg7087	:=	bOpcMsg_W[87];
	MM2VIS.bMsg7088	:=	bOpcMsg_W[88];
	MM2VIS.bMsg7089	:=	bOpcMsg_W[89];
	MM2VIS.bMsg7090	:=	bOpcMsg_W[90];
	MM2VIS.bMsg7091	:=	bOpcMsg_W[91];
	MM2VIS.bMsg7092	:=	bOpcMsg_W[92];
	MM2VIS.bMsg7093	:=	bOpcMsg_W[93];
	MM2VIS.bMsg7094	:=	bOpcMsg_W[94];
	MM2VIS.bMsg7095	:=	bOpcMsg_W[95];
	MM2VIS.bMsg7096	:=	bOpcMsg_W[96];
	MM2VIS.bMsg7097	:=	bOpcMsg_W[97];
	MM2VIS.bMsg7098	:=	bOpcMsg_W[98];
	MM2VIS.bMsg7099	:=	bOpcMsg_W[99];
	MM2VIS.bMsg7100	:=	bOpcMsg_W[100];
	MM2VIS.bMsg7101	:=	bOpcMsg_W[101];
	MM2VIS.bMsg7102	:=	bOpcMsg_W[102];
	MM2VIS.bMsg7103	:=	bOpcMsg_W[103];
	MM2VIS.bMsg7104	:=	bOpcMsg_W[104];
	MM2VIS.bMsg7105	:=	bOpcMsg_W[105];
	MM2VIS.bMsg7106	:=	bOpcMsg_W[106];
	MM2VIS.bMsg7107	:=	bOpcMsg_W[107];
	MM2VIS.bMsg7108	:=	bOpcMsg_W[108];
	MM2VIS.bMsg7109	:=	bOpcMsg_W[109];
	MM2VIS.bMsg7110	:=	bOpcMsg_W[110];
	MM2VIS.bMsg7111	:=	bOpcMsg_W[111];
	MM2VIS.bMsg7112	:=	bOpcMsg_W[112];
	MM2VIS.bMsg7113	:=	bOpcMsg_W[113];
	MM2VIS.bMsg7114	:=	bOpcMsg_W[114];
	MM2VIS.bMsg7115	:=	bOpcMsg_W[115];
	MM2VIS.bMsg7116	:=	bOpcMsg_W[116];
	MM2VIS.bMsg7117	:=	bOpcMsg_W[117];
	MM2VIS.bMsg7118	:=	bOpcMsg_W[118];
	MM2VIS.bMsg7119	:=	bOpcMsg_W[119];
	MM2VIS.bMsg7120	:=	bOpcMsg_W[120];
	MM2VIS.bMsg7121	:=	bOpcMsg_W[121];
	MM2VIS.bMsg7122	:=	bOpcMsg_W[122];
	MM2VIS.bMsg7123	:=	bOpcMsg_W[123];
	MM2VIS.bMsg7124	:=	bOpcMsg_W[124];
	MM2VIS.bMsg7125	:=	bOpcMsg_W[125];
	MM2VIS.bMsg7126	:=	bOpcMsg_W[126];
	MM2VIS.bMsg7127	:=	bOpcMsg_W[127];
	MM2VIS.bMsg7128	:=	bOpcMsg_W[128];
	MM2VIS.bMsg7129	:=	bOpcMsg_W[129];
	MM2VIS.bMsg7130	:=	bOpcMsg_W[130];
	MM2VIS.bMsg7131	:=	bOpcMsg_W[131];
	MM2VIS.bMsg7132	:=	bOpcMsg_W[132];
	MM2VIS.bMsg7133	:=	bOpcMsg_W[133];
	MM2VIS.bMsg7134	:=	bOpcMsg_W[134];
	MM2VIS.bMsg7135	:=	bOpcMsg_W[135];
	MM2VIS.bMsg7136	:=	bOpcMsg_W[136];
	MM2VIS.bMsg7137	:=	bOpcMsg_W[137];
	MM2VIS.bMsg7138	:=	bOpcMsg_W[138];
	MM2VIS.bMsg7139	:=	bOpcMsg_W[139];
	MM2VIS.bMsg7140	:=	bOpcMsg_W[140];
	MM2VIS.bMsg7141	:=	bOpcMsg_W[141];
	MM2VIS.bMsg7142	:=	bOpcMsg_W[142];
	MM2VIS.bMsg7143	:=	bOpcMsg_W[143];
	MM2VIS.bMsg7144	:=	bOpcMsg_W[144];
	MM2VIS.bMsg7145	:=	bOpcMsg_W[145];
	MM2VIS.bMsg7146	:=	bOpcMsg_W[146];
	MM2VIS.bMsg7147	:=	bOpcMsg_W[147];
	MM2VIS.bMsg7148	:=	bOpcMsg_W[148];
	MM2VIS.bMsg7149	:=	bOpcMsg_W[149];
	MM2VIS.bMsg7150	:=	bOpcMsg_W[150];
	MM2VIS.bMsg7151	:=	bOpcMsg_W[151];
	MM2VIS.bMsg7152	:=	bOpcMsg_W[152];
	MM2VIS.bMsg7153	:=	bOpcMsg_W[153];
	MM2VIS.bMsg7154	:=	bOpcMsg_W[154];
	MM2VIS.bMsg7155	:=	bOpcMsg_W[155];
	MM2VIS.bMsg7156	:=	bOpcMsg_W[156];
	MM2VIS.bMsg7157	:=	bOpcMsg_W[157];
	MM2VIS.bMsg7158	:=	bOpcMsg_W[158];
	MM2VIS.bMsg7159	:=	bOpcMsg_W[159];
	MM2VIS.bMsg7160	:=	bOpcMsg_W[160];
	MM2VIS.bMsg7161	:=	bOpcMsg_W[161];
	MM2VIS.bMsg7162	:=	bOpcMsg_W[162];
	MM2VIS.bMsg7163	:=	bOpcMsg_W[163];
	MM2VIS.bMsg7164	:=	bOpcMsg_W[164];
	MM2VIS.bMsg7165	:=	bOpcMsg_W[165];
	MM2VIS.bMsg7166	:=	bOpcMsg_W[166];
	MM2VIS.bMsg7167	:=	bOpcMsg_W[167];
	MM2VIS.bMsg7168	:=	bOpcMsg_W[168];
	MM2VIS.bMsg7169	:=	bOpcMsg_W[169];
	MM2VIS.bMsg7170	:=	bOpcMsg_W[170];
	MM2VIS.bMsg7171	:=	bOpcMsg_W[171];
	MM2VIS.bMsg7172	:=	bOpcMsg_W[172];
	MM2VIS.bMsg7173	:=	bOpcMsg_W[173];
	MM2VIS.bMsg7174	:=	bOpcMsg_W[174];
	MM2VIS.bMsg7175	:=	bOpcMsg_W[175];
	MM2VIS.bMsg7176	:=	bOpcMsg_W[176];
	MM2VIS.bMsg7177	:=	bOpcMsg_W[177];
	MM2VIS.bMsg7178	:=	bOpcMsg_W[178];
	MM2VIS.bMsg7179	:=	bOpcMsg_W[179];
	MM2VIS.bMsg7180	:=	bOpcMsg_W[180];
	MM2VIS.bMsg7181	:=	bOpcMsg_W[181];
	MM2VIS.bMsg7182	:=	bOpcMsg_W[182];
	MM2VIS.bMsg7183	:=	bOpcMsg_W[183];
	MM2VIS.bMsg7184	:=	bOpcMsg_W[184];
	MM2VIS.bMsg7185	:=	bOpcMsg_W[185];
	MM2VIS.bMsg7186	:=	bOpcMsg_W[186];
	MM2VIS.bMsg7187	:=	bOpcMsg_W[187];
	MM2VIS.bMsg7188	:=	bOpcMsg_W[188];
	MM2VIS.bMsg7189	:=	bOpcMsg_W[189];
	MM2VIS.bMsg7190	:=	bOpcMsg_W[190];
	MM2VIS.bMsg7191	:=	bOpcMsg_W[191];
	MM2VIS.bMsg7192	:=	bOpcMsg_W[192];
	MM2VIS.bMsg7193	:=	bOpcMsg_W[193];
	MM2VIS.bMsg7194	:=	bOpcMsg_W[194];
	MM2VIS.bMsg7195	:=	bOpcMsg_W[195];
	MM2VIS.bMsg7196	:=	bOpcMsg_W[196];
	MM2VIS.bMsg7197	:=	bOpcMsg_W[197];
	MM2VIS.bMsg7198	:=	bOpcMsg_W[198];
	MM2VIS.bMsg7199	:=	bOpcMsg_W[199];
	MM2VIS.bMsg7200	:=	bOpcMsg_W[200];
	MM2VIS.bMsg7201	:=	bOpcMsg_W[201];
	MM2VIS.bMsg7202	:=	bOpcMsg_W[202];
	MM2VIS.bMsg7203	:=	bOpcMsg_W[203];
	MM2VIS.bMsg7204	:=	bOpcMsg_W[204];
	MM2VIS.bMsg7205	:=	bOpcMsg_W[205];
	MM2VIS.bMsg7206	:=	bOpcMsg_W[206];
	MM2VIS.bMsg7207	:=	bOpcMsg_W[207];
	MM2VIS.bMsg7208	:=	bOpcMsg_W[208];
	MM2VIS.bMsg7209	:=	bOpcMsg_W[209];
	MM2VIS.bMsg7210	:=	bOpcMsg_W[210];
	MM2VIS.bMsg7211	:=	bOpcMsg_W[211];
	MM2VIS.bMsg7212	:=	bOpcMsg_W[212];
	MM2VIS.bMsg7213	:=	bOpcMsg_W[213];
	MM2VIS.bMsg7214	:=	bOpcMsg_W[214];
	MM2VIS.bMsg7215	:=	bOpcMsg_W[215];
	MM2VIS.bMsg7216	:=	bOpcMsg_W[216];
	MM2VIS.bMsg7217	:=	bOpcMsg_W[217];
	MM2VIS.bMsg7218	:=	bOpcMsg_W[218];
	MM2VIS.bMsg7219	:=	bOpcMsg_W[219];
	MM2VIS.bMsg7220	:=	bOpcMsg_W[220];
	MM2VIS.bMsg7221	:=	bOpcMsg_W[221];
	MM2VIS.bMsg7222	:=	bOpcMsg_W[222];
	MM2VIS.bMsg7223	:=	bOpcMsg_W[223];
	MM2VIS.bMsg7224	:=	bOpcMsg_W[224];
	MM2VIS.bMsg7225	:=	bOpcMsg_W[225];
	MM2VIS.bMsg7226	:=	bOpcMsg_W[226];
	MM2VIS.bMsg7227	:=	bOpcMsg_W[227];
	MM2VIS.bMsg7228	:=	bOpcMsg_W[228];
	MM2VIS.bMsg7229	:=	bOpcMsg_W[229];
	MM2VIS.bMsg7230	:=	bOpcMsg_W[230];
	MM2VIS.bMsg7231	:=	bOpcMsg_W[231];
	MM2VIS.bMsg7232	:=	bOpcMsg_W[232];
	MM2VIS.bMsg7233	:=	bOpcMsg_W[233];
	MM2VIS.bMsg7234	:=	bOpcMsg_W[234];
	MM2VIS.bMsg7235	:=	bOpcMsg_W[235];
	MM2VIS.bMsg7236	:=	bOpcMsg_W[236];
	MM2VIS.bMsg7237	:=	bOpcMsg_W[237];
	MM2VIS.bMsg7238	:=	bOpcMsg_W[238];
	MM2VIS.bMsg7239	:=	bOpcMsg_W[239];
	MM2VIS.bMsg7240	:=	bOpcMsg_W[240];
	MM2VIS.bMsg7241	:=	bOpcMsg_W[241];
	MM2VIS.bMsg7242	:=	bOpcMsg_W[242];
	MM2VIS.bMsg7243	:=	bOpcMsg_W[243];
	MM2VIS.bMsg7244	:=	bOpcMsg_W[244];
	MM2VIS.bMsg7245	:=	bOpcMsg_W[245];
	MM2VIS.bMsg7246	:=	bOpcMsg_W[246];
	MM2VIS.bMsg7247	:=	bOpcMsg_W[247];
	MM2VIS.bMsg7248	:=	bOpcMsg_W[248];
	MM2VIS.bMsg7249	:=	bOpcMsg_W[249];
	MM2VIS.bMsg7250	:=	bOpcMsg_W[250];
	MM2VIS.bMsg7251	:=	bOpcMsg_W[251];
	MM2VIS.bMsg7252	:=	bOpcMsg_W[252];
	MM2VIS.bMsg7253	:=	bOpcMsg_W[253];
	MM2VIS.bMsg7254	:=	bOpcMsg_W[254];
	MM2VIS.bMsg7255	:=	bOpcMsg_W[255];
	MM2VIS.bMsg7256	:=	bOpcMsg_W[256];
	MM2VIS.bMsg7257	:=	bOpcMsg_W[257];
	MM2VIS.bMsg7258	:=	bOpcMsg_W[258];
	MM2VIS.bMsg7259	:=	bOpcMsg_W[259];
	MM2VIS.bMsg7260	:=	bOpcMsg_W[260];
	MM2VIS.bMsg7261	:=	bOpcMsg_W[261];
	MM2VIS.bMsg7262	:=	bOpcMsg_W[262];
	MM2VIS.bMsg7263	:=	bOpcMsg_W[263];
	MM2VIS.bMsg7264	:=	bOpcMsg_W[264];
	MM2VIS.bMsg7265	:=	bOpcMsg_W[265];
	MM2VIS.bMsg7266	:=	bOpcMsg_W[266];
	MM2VIS.bMsg7267	:=	bOpcMsg_W[267];
	MM2VIS.bMsg7268	:=	bOpcMsg_W[268];
	MM2VIS.bMsg7269	:=	bOpcMsg_W[269];
	MM2VIS.bMsg7270	:=	bOpcMsg_W[270];
	MM2VIS.bMsg7271	:=	bOpcMsg_W[271];
	MM2VIS.bMsg7272	:=	bOpcMsg_W[272];
	MM2VIS.bMsg7273	:=	bOpcMsg_W[273];
	MM2VIS.bMsg7274	:=	bOpcMsg_W[274];
	MM2VIS.bMsg7275	:=	bOpcMsg_W[275];
	MM2VIS.bMsg7276	:=	bOpcMsg_W[276];
	MM2VIS.bMsg7277	:=	bOpcMsg_W[277];
	MM2VIS.bMsg7278	:=	bOpcMsg_W[278];
	MM2VIS.bMsg7279	:=	bOpcMsg_W[279];
	MM2VIS.bMsg7280	:=	bOpcMsg_W[280];
	MM2VIS.bMsg7281	:=	bOpcMsg_W[281];
	MM2VIS.bMsg7282	:=	bOpcMsg_W[282];
	MM2VIS.bMsg7283	:=	bOpcMsg_W[283];
	MM2VIS.bMsg7284	:=	bOpcMsg_W[284];
	MM2VIS.bMsg7285	:=	bOpcMsg_W[285];
	MM2VIS.bMsg7286	:=	bOpcMsg_W[286];
	MM2VIS.bMsg7287	:=	bOpcMsg_W[287];
	MM2VIS.bMsg7288	:=	bOpcMsg_W[288];
	MM2VIS.bMsg7289	:=	bOpcMsg_W[289];
	MM2VIS.bMsg7290	:=	bOpcMsg_W[290];
	MM2VIS.bMsg7291	:=	bOpcMsg_W[291];
	MM2VIS.bMsg7292	:=	bOpcMsg_W[292];
	MM2VIS.bMsg7293	:=	bOpcMsg_W[293];
	MM2VIS.bMsg7294	:=	bOpcMsg_W[294];
	MM2VIS.bMsg7295	:=	bOpcMsg_W[295];
	MM2VIS.bMsg7296	:=	bOpcMsg_W[296];
	MM2VIS.bMsg7297	:=	bOpcMsg_W[297];
	MM2VIS.bMsg7298	:=	bOpcMsg_W[298];
	MM2VIS.bMsg7299	:=	bOpcMsg_W[299];
	MM2VIS.bMsg7300	:=	bOpcMsg_W[300];
	MM2VIS.bMsg7301	:=	bOpcMsg_W[301];
	MM2VIS.bMsg7302	:=	bOpcMsg_W[302];
	MM2VIS.bMsg7303	:=	bOpcMsg_W[303];
	MM2VIS.bMsg7304	:=	bOpcMsg_W[304];
	MM2VIS.bMsg7305	:=	bOpcMsg_W[305];
	MM2VIS.bMsg7306	:=	bOpcMsg_W[306];
	MM2VIS.bMsg7307	:=	bOpcMsg_W[307];
	MM2VIS.bMsg7308	:=	bOpcMsg_W[308];
	MM2VIS.bMsg7309	:=	bOpcMsg_W[309];
	MM2VIS.bMsg7310	:=	bOpcMsg_W[310];
	MM2VIS.bMsg7311	:=	bOpcMsg_W[311];
	MM2VIS.bMsg7312	:=	bOpcMsg_W[312];
	MM2VIS.bMsg7313	:=	bOpcMsg_W[313];
	MM2VIS.bMsg7314	:=	bOpcMsg_W[314];
	MM2VIS.bMsg7315	:=	bOpcMsg_W[315];
	MM2VIS.bMsg7316	:=	bOpcMsg_W[316];
	MM2VIS.bMsg7317	:=	bOpcMsg_W[317];
	MM2VIS.bMsg7318	:=	bOpcMsg_W[318];
	MM2VIS.bMsg7319	:=	bOpcMsg_W[319];
	MM2VIS.bMsg7320	:=	bOpcMsg_W[320];
	MM2VIS.bMsg7321	:=	bOpcMsg_W[321];
	MM2VIS.bMsg7322	:=	bOpcMsg_W[322];
	MM2VIS.bMsg7323	:=	bOpcMsg_W[323];
	MM2VIS.bMsg7324	:=	bOpcMsg_W[324];
	MM2VIS.bMsg7325	:=	bOpcMsg_W[325];
	MM2VIS.bMsg7326	:=	bOpcMsg_W[326];
	MM2VIS.bMsg7327	:=	bOpcMsg_W[327];
	MM2VIS.bMsg7328	:=	bOpcMsg_W[328];
	MM2VIS.bMsg7329	:=	bOpcMsg_W[329];
	MM2VIS.bMsg7330	:=	bOpcMsg_W[330];
	MM2VIS.bMsg7331	:=	bOpcMsg_W[331];
	MM2VIS.bMsg7332	:=	bOpcMsg_W[332];
	MM2VIS.bMsg7333	:=	bOpcMsg_W[333];
	MM2VIS.bMsg7334	:=	bOpcMsg_W[334];
	MM2VIS.bMsg7335	:=	bOpcMsg_W[335];
	MM2VIS.bMsg7336	:=	bOpcMsg_W[336];
	MM2VIS.bMsg7337	:=	bOpcMsg_W[337];
	MM2VIS.bMsg7338	:=	bOpcMsg_W[338];
	MM2VIS.bMsg7339	:=	bOpcMsg_W[339];
	MM2VIS.bMsg7340	:=	bOpcMsg_W[340];
	MM2VIS.bMsg7341	:=	bOpcMsg_W[341];
	MM2VIS.bMsg7342	:=	bOpcMsg_W[342];
	MM2VIS.bMsg7343	:=	bOpcMsg_W[343];
	MM2VIS.bMsg7344	:=	bOpcMsg_W[344];
	MM2VIS.bMsg7345	:=	bOpcMsg_W[345];
	MM2VIS.bMsg7346	:=	bOpcMsg_W[346];
	MM2VIS.bMsg7347	:=	bOpcMsg_W[347];
	MM2VIS.bMsg7348	:=	bOpcMsg_W[348];
	MM2VIS.bMsg7349	:=	bOpcMsg_W[349];
	MM2VIS.bMsg7350	:=	bOpcMsg_W[350];
	MM2VIS.bMsg7351	:=	bOpcMsg_W[351];
	MM2VIS.bMsg7352	:=	bOpcMsg_W[352];
	MM2VIS.bMsg7353	:=	bOpcMsg_W[353];
	MM2VIS.bMsg7354	:=	bOpcMsg_W[354];
	MM2VIS.bMsg7355	:=	bOpcMsg_W[355];
	MM2VIS.bMsg7356	:=	bOpcMsg_W[356];
	MM2VIS.bMsg7357	:=	bOpcMsg_W[357];
	MM2VIS.bMsg7358	:=	bOpcMsg_W[358];
	MM2VIS.bMsg7359	:=	bOpcMsg_W[359];
	MM2VIS.bMsg7360	:=	bOpcMsg_W[360];
	MM2VIS.bMsg7361	:=	bOpcMsg_W[361];
	MM2VIS.bMsg7362	:=	bOpcMsg_W[362];
	MM2VIS.bMsg7363	:=	bOpcMsg_W[363];
	MM2VIS.bMsg7364	:=	bOpcMsg_W[364];
	MM2VIS.bMsg7365	:=	bOpcMsg_W[365];
	MM2VIS.bMsg7366	:=	bOpcMsg_W[366];
	MM2VIS.bMsg7367	:=	bOpcMsg_W[367];
	MM2VIS.bMsg7368	:=	bOpcMsg_W[368];
	MM2VIS.bMsg7369	:=	bOpcMsg_W[369];
	MM2VIS.bMsg7370	:=	bOpcMsg_W[370];
	MM2VIS.bMsg7371	:=	bOpcMsg_W[371];
	MM2VIS.bMsg7372	:=	bOpcMsg_W[372];
	MM2VIS.bMsg7373	:=	bOpcMsg_W[373];
	MM2VIS.bMsg7374	:=	bOpcMsg_W[374];
	MM2VIS.bMsg7375	:=	bOpcMsg_W[375];
	MM2VIS.bMsg7376	:=	bOpcMsg_W[376];
	MM2VIS.bMsg7377	:=	bOpcMsg_W[377];
	MM2VIS.bMsg7378	:=	bOpcMsg_W[378];
	MM2VIS.bMsg7379	:=	bOpcMsg_W[379];
	MM2VIS.bMsg7380	:=	bOpcMsg_W[380];
	MM2VIS.bMsg7381	:=	bOpcMsg_W[381];
	MM2VIS.bMsg7382	:=	bOpcMsg_W[382];
	MM2VIS.bMsg7383	:=	bOpcMsg_W[383];
	MM2VIS.bMsg7384	:=	bOpcMsg_W[384];
	MM2VIS.bMsg7385	:=	bOpcMsg_W[385];
	MM2VIS.bMsg7386	:=	bOpcMsg_W[386];
	MM2VIS.bMsg7387	:=	bOpcMsg_W[387];
	MM2VIS.bMsg7388	:=	bOpcMsg_W[388];
	MM2VIS.bMsg7389	:=	bOpcMsg_W[389];
	MM2VIS.bMsg7390	:=	bOpcMsg_W[390];
	MM2VIS.bMsg7391	:=	bOpcMsg_W[391];
	MM2VIS.bMsg7392	:=	bOpcMsg_W[392];
	MM2VIS.bMsg7393	:=	bOpcMsg_W[393];
	MM2VIS.bMsg7394	:=	bOpcMsg_W[394];
	MM2VIS.bMsg7395	:=	bOpcMsg_W[395];
	MM2VIS.bMsg7396	:=	bOpcMsg_W[396];
	MM2VIS.bMsg7397	:=	bOpcMsg_W[397];
	MM2VIS.bMsg7398	:=	bOpcMsg_W[398];
	MM2VIS.bMsg7399	:=	bOpcMsg_W[399];
	MM2VIS.bMsg7400	:=	bOpcMsg_W[400];
	MM2VIS.bMsg7401	:=	bOpcMsg_W[401];
	MM2VIS.bMsg7402	:=	bOpcMsg_W[402];
	MM2VIS.bMsg7403	:=	bOpcMsg_W[403];
	MM2VIS.bMsg7404	:=	bOpcMsg_W[404];
	MM2VIS.bMsg7405	:=	bOpcMsg_W[405];
	MM2VIS.bMsg7406	:=	bOpcMsg_W[406];
	MM2VIS.bMsg7407	:=	bOpcMsg_W[407];
	MM2VIS.bMsg7408	:=	bOpcMsg_W[408];
	MM2VIS.bMsg7409	:=	bOpcMsg_W[409];
	MM2VIS.bMsg7410	:=	bOpcMsg_W[410];
	MM2VIS.bMsg7411	:=	bOpcMsg_W[411];
	MM2VIS.bMsg7412	:=	bOpcMsg_W[412];
	MM2VIS.bMsg7413	:=	bOpcMsg_W[413];
	MM2VIS.bMsg7414	:=	bOpcMsg_W[414];
	MM2VIS.bMsg7415	:=	bOpcMsg_W[415];
	MM2VIS.bMsg7416	:=	bOpcMsg_W[416];
	MM2VIS.bMsg7417	:=	bOpcMsg_W[417];
	MM2VIS.bMsg7418	:=	bOpcMsg_W[418];
	MM2VIS.bMsg7419	:=	bOpcMsg_W[419];
	MM2VIS.bMsg7420	:=	bOpcMsg_W[420];
	MM2VIS.bMsg7421	:=	bOpcMsg_W[421];
	MM2VIS.bMsg7422	:=	bOpcMsg_W[422];
	MM2VIS.bMsg7423	:=	bOpcMsg_W[423];
	MM2VIS.bMsg7424	:=	bOpcMsg_W[424];
	MM2VIS.bMsg7425	:=	bOpcMsg_W[425];
	MM2VIS.bMsg7426	:=	bOpcMsg_W[426];
	MM2VIS.bMsg7427	:=	bOpcMsg_W[427];
	MM2VIS.bMsg7428	:=	bOpcMsg_W[428];
	MM2VIS.bMsg7429	:=	bOpcMsg_W[429];
	MM2VIS.bMsg7430	:=	bOpcMsg_W[430];
	MM2VIS.bMsg7431	:=	bOpcMsg_W[431];
	MM2VIS.bMsg7432	:=	bOpcMsg_W[432];
	MM2VIS.bMsg7433	:=	bOpcMsg_W[433];
	MM2VIS.bMsg7434	:=	bOpcMsg_W[434];
	MM2VIS.bMsg7435	:=	bOpcMsg_W[435];
	MM2VIS.bMsg7436	:=	bOpcMsg_W[436];
	MM2VIS.bMsg7437	:=	bOpcMsg_W[437];
	MM2VIS.bMsg7438	:=	bOpcMsg_W[438];
	MM2VIS.bMsg7439	:=	bOpcMsg_W[439];
	MM2VIS.bMsg7440	:=	bOpcMsg_W[440];
	MM2VIS.bMsg7441	:=	bOpcMsg_W[441];
	MM2VIS.bMsg7442	:=	bOpcMsg_W[442];
	MM2VIS.bMsg7443	:=	bOpcMsg_W[443];
	MM2VIS.bMsg7444	:=	bOpcMsg_W[444];
	MM2VIS.bMsg7445	:=	bOpcMsg_W[445];
	MM2VIS.bMsg7446	:=	bOpcMsg_W[446];
	MM2VIS.bMsg7447	:=	bOpcMsg_W[447];
	MM2VIS.bMsg7448	:=	bOpcMsg_W[448];
	MM2VIS.bMsg7449	:=	bOpcMsg_W[449];
	MM2VIS.bMsg7450	:=	bOpcMsg_W[450];
	MM2VIS.bMsg7451	:=	bOpcMsg_W[451];
	MM2VIS.bMsg7452	:=	bOpcMsg_W[452];
	MM2VIS.bMsg7453	:=	bOpcMsg_W[453];
	MM2VIS.bMsg7454	:=	bOpcMsg_W[454];
	MM2VIS.bMsg7455	:=	bOpcMsg_W[455];
	MM2VIS.bMsg7456	:=	bOpcMsg_W[456];
	MM2VIS.bMsg7457	:=	bOpcMsg_W[457];
	MM2VIS.bMsg7458	:=	bOpcMsg_W[458];
	MM2VIS.bMsg7459	:=	bOpcMsg_W[459];
	MM2VIS.bMsg7460	:=	bOpcMsg_W[460];
	MM2VIS.bMsg7461	:=	bOpcMsg_W[461];
	MM2VIS.bMsg7462	:=	bOpcMsg_W[462];
	MM2VIS.bMsg7463	:=	bOpcMsg_W[463];
	MM2VIS.bMsg7464	:=	bOpcMsg_W[464];
	MM2VIS.bMsg7465	:=	bOpcMsg_W[465];
	MM2VIS.bMsg7466	:=	bOpcMsg_W[466];
	MM2VIS.bMsg7467	:=	bOpcMsg_W[467];
	MM2VIS.bMsg7468	:=	bOpcMsg_W[468];
	MM2VIS.bMsg7469	:=	bOpcMsg_W[469];
	MM2VIS.bMsg7470	:=	bOpcMsg_W[470];
	MM2VIS.bMsg7471	:=	bOpcMsg_W[471];
	MM2VIS.bMsg7472	:=	bOpcMsg_W[472];
	MM2VIS.bMsg7473	:=	bOpcMsg_W[473];
	MM2VIS.bMsg7474	:=	bOpcMsg_W[474];
	MM2VIS.bMsg7475	:=	bOpcMsg_W[475];
	MM2VIS.bMsg7476	:=	bOpcMsg_W[476];
	MM2VIS.bMsg7477	:=	bOpcMsg_W[477];
	MM2VIS.bMsg7478	:=	bOpcMsg_W[478];
	MM2VIS.bMsg7479	:=	bOpcMsg_W[479];
	MM2VIS.bMsg7480	:=	bOpcMsg_W[480];
	MM2VIS.bMsg7481	:=	bOpcMsg_W[481];
	MM2VIS.bMsg7482	:=	bOpcMsg_W[482];
	MM2VIS.bMsg7483	:=	bOpcMsg_W[483];
	MM2VIS.bMsg7484	:=	bOpcMsg_W[484];
	MM2VIS.bMsg7485	:=	bOpcMsg_W[485];
	MM2VIS.bMsg7486	:=	bOpcMsg_W[486];
	MM2VIS.bMsg7487	:=	bOpcMsg_W[487];
	MM2VIS.bMsg7488	:=	bOpcMsg_W[488];
	MM2VIS.bMsg7489	:=	bOpcMsg_W[489];
	MM2VIS.bMsg7490	:=	bOpcMsg_W[490];
	MM2VIS.bMsg7491	:=	bOpcMsg_W[491];
	MM2VIS.bMsg7492	:=	bOpcMsg_W[492];
	MM2VIS.bMsg7493	:=	bOpcMsg_W[493];
	MM2VIS.bMsg7494	:=	bOpcMsg_W[494];
	MM2VIS.bMsg7495	:=	bOpcMsg_W[495];
	MM2VIS.bMsg7496	:=	bOpcMsg_W[496];
	MM2VIS.bMsg7497	:=	bOpcMsg_W[497];
	MM2VIS.bMsg7498	:=	bOpcMsg_W[498];
	MM2VIS.bMsg7499	:=	bOpcMsg_W[499];
	MM2VIS.bMsg7500	:=	bOpcMsg_W[500];
	MM2VIS.bMsg7501	:=	bOpcMsg_W[501];
	MM2VIS.bMsg7502	:=	bOpcMsg_W[502];
	MM2VIS.bMsg7503	:=	bOpcMsg_W[503];
	MM2VIS.bMsg7504	:=	bOpcMsg_W[504];
	MM2VIS.bMsg7505	:=	bOpcMsg_W[505];
	MM2VIS.bMsg7506	:=	bOpcMsg_W[506];
	MM2VIS.bMsg7507	:=	bOpcMsg_W[507];
	MM2VIS.bMsg7508	:=	bOpcMsg_W[508];
	MM2VIS.bMsg7509	:=	bOpcMsg_W[509];
	MM2VIS.bMsg7510	:=	bOpcMsg_W[510];
	MM2VIS.bMsg7511	:=	bOpcMsg_W[511];
	MM2VIS.bMsg7512	:=	bOpcMsg_W[512];
	MM2VIS.bMsg7513	:=	bOpcMsg_W[513];
	MM2VIS.bMsg7514	:=	bOpcMsg_W[514];
	MM2VIS.bMsg7515	:=	bOpcMsg_W[515];
	MM2VIS.bMsg7516	:=	bOpcMsg_W[516];
	MM2VIS.bMsg7517	:=	bOpcMsg_W[517];
	MM2VIS.bMsg7518	:=	bOpcMsg_W[518];
	MM2VIS.bMsg7519	:=	bOpcMsg_W[519];
	MM2VIS.bMsg7520	:=	bOpcMsg_W[520];
	MM2VIS.bMsg7521	:=	bOpcMsg_W[521];
	MM2VIS.bMsg7522	:=	bOpcMsg_W[522];
	MM2VIS.bMsg7523	:=	bOpcMsg_W[523];
	MM2VIS.bMsg7524	:=	bOpcMsg_W[524];
	MM2VIS.bMsg7525	:=	bOpcMsg_W[525];
	MM2VIS.bMsg7526	:=	bOpcMsg_W[526];
	MM2VIS.bMsg7527	:=	bOpcMsg_W[527];
	MM2VIS.bMsg7528	:=	bOpcMsg_W[528];
	MM2VIS.bMsg7529	:=	bOpcMsg_W[529];
	MM2VIS.bMsg7530	:=	bOpcMsg_W[530];

	MM2VIS.bMsg7600	:=	bOpcMsg_W[600];
	MM2VIS.bMsg7601	:=	bOpcMsg_W[601];
	MM2VIS.bMsg7602	:=	bOpcMsg_W[602];
	MM2VIS.bMsg7603	:=	bOpcMsg_W[603];
	MM2VIS.bMsg7604	:=	bOpcMsg_W[604];
	MM2VIS.bMsg7605	:=	bOpcMsg_W[605];
	MM2VIS.bMsg7606	:=	bOpcMsg_W[606];
	MM2VIS.bMsg7607	:=	bOpcMsg_W[607];
	MM2VIS.bMsg7608	:=	bOpcMsg_W[608];
	MM2VIS.bMsg7609	:=	bOpcMsg_W[609];
	MM2VIS.bMsg7610	:=	bOpcMsg_W[610];
	MM2VIS.bMsg7611	:=	bOpcMsg_W[611];
	MM2VIS.bMsg7612	:=	bOpcMsg_W[612];
	MM2VIS.bMsg7613	:=	bOpcMsg_W[613];
	MM2VIS.bMsg7614	:=	bOpcMsg_W[614];
	MM2VIS.bMsg7615	:=	bOpcMsg_W[615];
	MM2VIS.bMsg7616	:=	bOpcMsg_W[616];
	MM2VIS.bMsg7617	:=	bOpcMsg_W[617];
	MM2VIS.bMsg7618	:=	bOpcMsg_W[618];
	MM2VIS.bMsg7619	:=	bOpcMsg_W[619];
	MM2VIS.bMsg7620	:=	bOpcMsg_W[620];
	MM2VIS.bMsg7621	:=	bOpcMsg_W[621];
	MM2VIS.bMsg7622	:=	bOpcMsg_W[622];
	MM2VIS.bMsg7623	:=	bOpcMsg_W[623];
	MM2VIS.bMsg7624	:=	bOpcMsg_W[624];
	MM2VIS.bMsg7625	:=	bOpcMsg_W[625];
	MM2VIS.bMsg7626	:=	bOpcMsg_W[626];
	MM2VIS.bMsg7627	:=	bOpcMsg_W[627];
	MM2VIS.bMsg7628	:=	bOpcMsg_W[628];
	MM2VIS.bMsg7629	:=	bOpcMsg_W[629];
	MM2VIS.bMsg7630	:=	bOpcMsg_W[630];
	MM2VIS.bMsg7631	:=	bOpcMsg_W[631];
	MM2VIS.bMsg7632	:=	bOpcMsg_W[632];
	MM2VIS.bMsg7633	:=	bOpcMsg_W[633];
	MM2VIS.bMsg7634	:=	bOpcMsg_W[634];
	MM2VIS.bMsg7635	:=	bOpcMsg_W[635];
	MM2VIS.bMsg7636	:=	bOpcMsg_W[636];
	MM2VIS.bMsg7637	:=	bOpcMsg_W[637];
	MM2VIS.bMsg7638	:=	bOpcMsg_W[638];
	MM2VIS.bMsg7639	:=	bOpcMsg_W[639];
	MM2VIS.bMsg7640	:=	bOpcMsg_W[640];
	MM2VIS.bMsg7641	:=	bOpcMsg_W[641];
	MM2VIS.bMsg7642	:=	bOpcMsg_W[642];
	MM2VIS.bMsg7643	:=	bOpcMsg_W[643];
	MM2VIS.bMsg7644	:=	bOpcMsg_W[644];
	MM2VIS.bMsg7645	:=	bOpcMsg_W[645];
	MM2VIS.bMsg7646	:=	bOpcMsg_W[646];
	MM2VIS.bMsg7647	:=	bOpcMsg_W[647];
	MM2VIS.bMsg7648	:=	bOpcMsg_W[648];
	MM2VIS.bMsg7649	:=	bOpcMsg_W[649];
	MM2VIS.bMsg7650	:=	bOpcMsg_W[650];
	MM2VIS.bMsg7651	:=	bOpcMsg_W[651];
	MM2VIS.bMsg7652	:=	bOpcMsg_W[652];
	MM2VIS.bMsg7653	:=	bOpcMsg_W[653];
	MM2VIS.bMsg7654	:=	bOpcMsg_W[654];
	MM2VIS.bMsg7655	:=	bOpcMsg_W[655];
	MM2VIS.bMsg7656	:=	bOpcMsg_W[656];
	MM2VIS.bMsg7657	:=	bOpcMsg_W[657];
	MM2VIS.bMsg7658	:=	bOpcMsg_W[658];
	MM2VIS.bMsg7659	:=	bOpcMsg_W[659];
	MM2VIS.bMsg7660	:=	bOpcMsg_W[660];

	MM2VIS.bMsg7700	:=	bOpcMsg_W[700];
	MM2VIS.bMsg7701	:=	bOpcMsg_W[701];
	MM2VIS.bMsg7702	:=	bOpcMsg_W[702];
	MM2VIS.bMsg7703	:=	bOpcMsg_W[703];
	MM2VIS.bMsg7704	:=	bOpcMsg_W[704];
	MM2VIS.bMsg7705	:=	bOpcMsg_W[705];
	MM2VIS.bMsg7706	:=	bOpcMsg_W[706];
	MM2VIS.bMsg7707	:=	bOpcMsg_W[707];
	MM2VIS.bMsg7708	:=	bOpcMsg_W[708];
	MM2VIS.bMsg7709	:=	bOpcMsg_W[709];
	MM2VIS.bMsg7710	:=	bOpcMsg_W[710];
	MM2VIS.bMsg7711	:=	bOpcMsg_W[711];
	MM2VIS.bMsg7712	:=	bOpcMsg_W[712];
	MM2VIS.bMsg7713	:=	bOpcMsg_W[713];
	MM2VIS.bMsg7714	:=	bOpcMsg_W[714];
	MM2VIS.bMsg7715	:=	bOpcMsg_W[715];
	MM2VIS.bMsg7716	:=	bOpcMsg_W[716];
	MM2VIS.bMsg7717	:=	bOpcMsg_W[717];
	MM2VIS.bMsg7718	:=	bOpcMsg_W[718];
	MM2VIS.bMsg7719	:=	bOpcMsg_W[719];
	MM2VIS.bMsg7720	:=	bOpcMsg_W[720];
	MM2VIS.bMsg7721	:=	bOpcMsg_W[721];
	MM2VIS.bMsg7722	:=	bOpcMsg_W[722];
	MM2VIS.bMsg7723	:=	bOpcMsg_W[723];
	MM2VIS.bMsg7724	:=	bOpcMsg_W[724];
	MM2VIS.bMsg7725	:=	bOpcMsg_W[725];
	MM2VIS.bMsg7726	:=	bOpcMsg_W[726];
	MM2VIS.bMsg7727	:=	bOpcMsg_W[727];
	MM2VIS.bMsg7728	:=	bOpcMsg_W[728];
	MM2VIS.bMsg7729	:=	bOpcMsg_W[729];
	MM2VIS.bMsg7730	:=	bOpcMsg_W[730];
	MM2VIS.bMsg7731	:=	bOpcMsg_W[731];
	MM2VIS.bMsg7732	:=	bOpcMsg_W[732];
	MM2VIS.bMsg7733	:=	bOpcMsg_W[733];
	MM2VIS.bMsg7734	:=	bOpcMsg_W[734];
	MM2VIS.bMsg7735	:=	bOpcMsg_W[735];
	MM2VIS.bMsg7736	:=	bOpcMsg_W[736];
	MM2VIS.bMsg7737	:=	bOpcMsg_W[737];
	MM2VIS.bMsg7738	:=	bOpcMsg_W[738];
	MM2VIS.bMsg7739	:=	bOpcMsg_W[739];
	MM2VIS.bMsg7740	:=	bOpcMsg_W[740];
	MM2VIS.bMsg7741	:=	bOpcMsg_W[741];
	MM2VIS.bMsg7742	:=	bOpcMsg_W[742];
	MM2VIS.bMsg7743	:=	bOpcMsg_W[743];
	MM2VIS.bMsg7744	:=	bOpcMsg_W[744];
	MM2VIS.bMsg7745	:=	bOpcMsg_W[745];
	MM2VIS.bMsg7746	:=	bOpcMsg_W[746];
	MM2VIS.bMsg7747	:=	bOpcMsg_W[747];
	MM2VIS.bMsg7748	:=	bOpcMsg_W[748];
	MM2VIS.bMsg7749	:=	bOpcMsg_W[749];
	MM2VIS.bMsg7750	:=	bOpcMsg_W[750];
	MM2VIS.bMsg7751	:=	bOpcMsg_W[751];
	MM2VIS.bMsg7752	:=	bOpcMsg_W[752];
	MM2VIS.bMsg7753	:=	bOpcMsg_W[753];
	MM2VIS.bMsg7754	:=	bOpcMsg_W[754];
	MM2VIS.bMsg7755	:=	bOpcMsg_W[755];
	MM2VIS.bMsg7756	:=	bOpcMsg_W[756];
	MM2VIS.bMsg7757	:=	bOpcMsg_W[757];
	MM2VIS.bMsg7758	:=	bOpcMsg_W[758];
	MM2VIS.bMsg7759	:=	bOpcMsg_W[759];
	MM2VIS.bMsg7760	:=	bOpcMsg_W[760];
	MM2VIS.bMsg7761	:=	bOpcMsg_W[761];
	MM2VIS.bMsg7762	:=	bOpcMsg_W[762];
	MM2VIS.bMsg7763	:=	bOpcMsg_W[763];
	MM2VIS.bMsg7764	:=	bOpcMsg_W[764];
	MM2VIS.bMsg7765	:=	bOpcMsg_W[765];
	MM2VIS.bMsg7766	:=	bOpcMsg_W[766];
	MM2VIS.bMsg7767	:=	bOpcMsg_W[767];
	MM2VIS.bMsg7768	:=	bOpcMsg_W[768];
	MM2VIS.bMsg7769	:=	bOpcMsg_W[769];
	MM2VIS.bMsg7770	:=	bOpcMsg_W[770];
	MM2VIS.bMsg7771	:=	bOpcMsg_W[771];
	MM2VIS.bMsg7772	:=	bOpcMsg_W[772];
	MM2VIS.bMsg7773	:=	bOpcMsg_W[773];
	MM2VIS.bMsg7774	:=	bOpcMsg_W[774];
	MM2VIS.bMsg7775	:=	bOpcMsg_W[775];
	MM2VIS.bMsg7776	:=	bOpcMsg_W[776];
	MM2VIS.bMsg7777	:=	bOpcMsg_W[777];
	MM2VIS.bMsg7778	:=	bOpcMsg_W[778];
	MM2VIS.bMsg7779	:=	bOpcMsg_W[779];
	MM2VIS.bMsg7780	:=	bOpcMsg_W[780];
	MM2VIS.bMsg7781	:=	bOpcMsg_W[781];
	MM2VIS.bMsg7782	:=	bOpcMsg_W[782];
	MM2VIS.bMsg7783	:=	bOpcMsg_W[783];
	MM2VIS.bMsg7784	:=	bOpcMsg_W[784];
	MM2VIS.bMsg7785	:=	bOpcMsg_W[785];
	MM2VIS.bMsg7786	:=	bOpcMsg_W[786];
	MM2VIS.bMsg7787	:=	bOpcMsg_W[787];
	MM2VIS.bMsg7788	:=	bOpcMsg_W[788];
	MM2VIS.bMsg7789	:=	bOpcMsg_W[789];
	MM2VIS.bMsg7790	:=	bOpcMsg_W[790];
	MM2VIS.bMsg7791	:=	bOpcMsg_W[791];
	MM2VIS.bMsg7792	:=	bOpcMsg_W[792];
	MM2VIS.bMsg7793	:=	bOpcMsg_W[793];
	MM2VIS.bMsg7794	:=	bOpcMsg_W[794];
	MM2VIS.bMsg7795	:=	bOpcMsg_W[795];
	MM2VIS.bMsg7796	:=	bOpcMsg_W[796];
	MM2VIS.bMsg7797	:=	bOpcMsg_W[797];
	MM2VIS.bMsg7798	:=	bOpcMsg_W[798];
	MM2VIS.bMsg7799	:=	bOpcMsg_W[799];
END_PROGRAM
```

### Program Logical/DataInterface/OpcVE (IEC) - OPC Var for Testbench

#### OpcVE.st
```iecst
(*******************************************************************************
OpcVE	 Variables read or write to Testbench

This code is confidential AND proprietary to the INNIO Company.
It may NOT be used in any form, or reproduced in any manner, without the express
written permission of the INNIO Company.
Copyright, INNIO Company, 2022

- list addidtional customized IO channels

Customized modifications: -
------------------------

History:
-------
V1.00.0	14.09.2022		Vockenberger	Neu erstellt
V1.01.0	31.05.2023		Vockenberger	Zusätzliche Jalousien eingefügt
		28.07.2023		Vockenberger	Struktur von OPC_DI geändert
V1.02.0	20.03.2024		Vockenberger	Kühlregister, Raumtemp. Variablen hinzugefügt
V1.03.0	09.01.2025		Gruber St.		cleanUp after change of parameter structure

Instructions FOR use:
--------------------

Outstandings:
------------

*******************************************************************************)

PROGRAM _CYCLIC

	(**Wird von Motor-CPU geschrieben**********************)
	(**REAL**)
	rOpcVE_R[0]		:=	VIS2MM.tCtr_ER_In.Y_man;
	rOpcVE_R[1]		:=	VIS2MM.tCtr_ER_In.X_min;
	rOpcVE_R[2]		:=	VIS2MM.tCtr_ER_In.X_max;
	rOpcVE_R[3]		:=	INT_TO_REAL(VIS2MM.tCtr_ER_In.Tune_quality);

	rOpcVE_R[4]		:=	VIS2MM.tCtr_OutlVE_RDP_In.Y_man;
	rOpcVE_R[5]		:=	VIS2MM.tCtr_OutlVE_RDP_In.X_min;
	rOpcVE_R[6]		:=	VIS2MM.tCtr_OutlVE_RDP_In.X_max;
	rOpcVE_R[7]		:=	INT_TO_REAL(VIS2MM.tCtr_OutlVE_RDP_In.Tune_quality);

	rOpcVE_R[8]		:=	VIS2MM.tCtr_IntakeAir_In.Y_man;
	rOpcVE_R[9]		:=	VIS2MM.tCtr_IntakeAir_In.X_min;
	rOpcVE_R[10]	:=	VIS2MM.tCtr_IntakeAir_In.X_max;
	rOpcVE_R[11]	:=	INT_TO_REAL(VIS2MM.tCtr_IntakeAir_In.Tune_quality);

	rOpcVE_R[12]	:=	IN_DI.rP_Act_Norm_Filt;
	rOpcVE_R[13]	:=	IN_DI.rP_Nom_Gastype[1];
	rOpcVE_R[14]	:=	IN_DI.rP_Nom_Gastype[2];
	rOpcVE_R[15]	:=	IN_DI.rP_Nom_Gastype[3];
	rOpcVE_R[16]	:=	Para.rT_CtrER_WexRun;
	rOpcVE_R[17]	:=	Para.rT_CtrER_WexStop;
	rOpcVE_R[18]	:=	Para.tCtr_OutlVE_RDP.W_set;
	rOpcVE_R[19]	:=	Para.tCtr_IntakeAir.W_set;
	rOpcVE_R[20];

	rOpcVE_R[21];
	rOpcVE_R[22];
	rOpcVE_R[23];
	rOpcVE_R[24];
	rOpcVE_R[25];
	rOpcVE_R[26];
	rOpcVE_R[27];
	rOpcVE_R[28];
	rOpcVE_R[29];
	rOpcVE_R[30];

	(**BOOL**)
	bOpcVE_R[0]	:=	VIS2MM.tCtr_ER_In.Y_man_Active;
	bOpcVE_R[1]	:=	VIS2MM.tCtr_ER_In.W_ext_Active;
	bOpcVE_R[2]	:=	VIS2MM.tCtr_ER_In.Tune_PI;
	bOpcVE_R[3]	:=	VIS2MM.tCtr_ER_In.Tune_PID;
	bOpcVE_R[4]	:=	VIS2MM.tCtr_ER_In.Tune_start;
	bOpcVE_R[5]	:=	VIS2MM.tCtr_ER_In.Tune_stop;
	bOpcVE_R[6]	:=	VIS2MM.tCtr_ER_In.Tune_takeover;

	bOpcVE_R[7]		:=	VIS2MM.tCtr_OutlVE_RDP_In.Y_man_Active;
	bOpcVE_R[8]		:=	VIS2MM.tCtr_OutlVE_RDP_In.W_ext_Active;
	bOpcVE_R[9]		:=	VIS2MM.tCtr_OutlVE_RDP_In.Tune_PI;
	bOpcVE_R[10]	:=	VIS2MM.tCtr_OutlVE_RDP_In.Tune_PID;
	bOpcVE_R[11]	:=	VIS2MM.tCtr_OutlVE_RDP_In.Tune_start;
	bOpcVE_R[12]	:=	VIS2MM.tCtr_OutlVE_RDP_In.Tune_stop;
	bOpcVE_R[13]	:=	VIS2MM.tCtr_OutlVE_RDP_In.Tune_takeover;

	bOpcVE_R[14]	:=	VIS2MM.tCtr_IntakeAir_In.Y_man_Active;
	bOpcVE_R[15]	:=	VIS2MM.tCtr_IntakeAir_In.W_ext_Active;
	bOpcVE_R[16]	:=	VIS2MM.tCtr_IntakeAir_In.Tune_PI;
	bOpcVE_R[17]	:=	VIS2MM.tCtr_IntakeAir_In.Tune_PID;
	bOpcVE_R[18]	:=	VIS2MM.tCtr_IntakeAir_In.Tune_start;
	bOpcVE_R[19]	:=	VIS2MM.tCtr_IntakeAir_In.Tune_stop;
	bOpcVE_R[20]	:=	VIS2MM.tCtr_IntakeAir_In.Tune_takeover;

	bOpcVE_R[21]	:=	VIS2MM.bDem_ERV_Aut_Vis;
	bOpcVE_R[22]	:=	VIS2MM.bCool_Air_Active;
	bOpcVE_R[23];
	bOpcVE_R[24];
	bOpcVE_R[25];
	bOpcVE_R[26];
	bOpcVE_R[27];
	bOpcVE_R[28];
	bOpcVE_R[29];
	bOpcVE_R[30];

	(*Ventilation from Testbench*)
	MM2VIS.rSet_InLou			:=	rOpcVE_W[0];
	MM2VIS.rSet_OutLou			:=	rOpcVE_W[1];
	MM2VIS.rSet_CircLou			:=	rOpcVE_W[2];
	MM2VIS.rSet_InLouEng		:=	rOpcVE_W[3];
	MM2VIS.rSet_CircLouEng		:=	rOpcVE_W[4];
	MM2VIS.rCtr_InER_FC			:=	rOpcVE_W[5];
	MM2VIS.rCtr_OutER_FC		:=	rOpcVE_W[6];
	MM2VIS.rCtr_InEngER_FC		:=	rOpcVE_W[7];
	MM2VIS.rCtr_CV_InAirHeat	:=	rOpcVE_W[8];
	MM2VIS.rCtr_CV_InAirCool	:=	rOpcVE_W[9];

	MM2VIS.rT_AirER_Avg			:=	rOpcVE_W[10];
	MM2VIS.rPos_InLouEng1 		:=	rOpcVE_W[11];
	MM2VIS.rPos_CircLouEng1		:=	rOpcVE_W[12];
	MM2VIS.rPos_CV_InAirHeat	:=	rOpcVE_W[13];
	MM2VIS.rPos_CV_InAirCool	:=	rOpcVE_W[14];
	MM2VIS.rT_AirER1			:=	rOpcVE_W[15];
	MM2VIS.rT_AirER2			:=	rOpcVE_W[16];
	MM2VIS.rT_AirER3			:=	rOpcVE_W[17];
	MM2VIS.rT_AirER4			:=	rOpcVE_W[18];
	MM2VIS.rT_AirOutdoor		:=	rOpcVE_W[19];

	MM2VIS.rT_FreshAirIn	:=	rOpcVE_W[20];
	MM2VIS.rT_FreshAirEng	:=	rOpcVE_W[21];
	MM2VIS.rT_HW_Air_Re		:=	rOpcVE_W[22];
	MM2VIS.rT_HW_Air_Su		:=	rOpcVE_W[23];
	MM2VIS.rPos_InlLou1		:=	rOpcVE_W[24];
	MM2VIS.rPos_InlLou2		:=	rOpcVE_W[25];
	MM2VIS.rPos_OutlLou1	:=	rOpcVE_W[26];
	MM2VIS.rPos_OutlLou2	:=	rOpcVE_W[27];
	MM2VIS.rPos_CircLou1	:=	rOpcVE_W[28];
	MM2VIS.rPos_CircLou2	:=	rOpcVE_W[29];

	MM2VIS.rPrDiff_ER		:=	rOpcVE_W[30];
	MM2VIS.rSet_InLouRoom	:=	rOpcVE_W[31];
	MM2VIS.rPos_OutlLou3	:=	rOpcVE_W[32];
	MM2VIS.rPos_OutlLou4	:=	rOpcVE_W[33];
	MM2VIS.rPos_InLouEng2	:=	rOpcVE_W[34];
	MM2VIS.rPos_CircLouEng2	:=	rOpcVE_W[35];
	MM2VIS.rPos_InlLouRoom1	:=	rOpcVE_W[36];
	MM2VIS.rPos_InlLouRoom2	:=	rOpcVE_W[37];
	MM2VIS.rPos_InlLouRoom3	:=	rOpcVE_W[38];
	MM2VIS.rPos_InlLouRoom4	:=	rOpcVE_W[39];

	MM2VIS.rPr_Cool_Air_Re	:=	rOpcVE_W[40];
	MM2VIS.rPr_HW_Air_Re	:=	rOpcVE_W[41];
	MM2VIS.rT_Cool_Air_Re	:=	rOpcVE_W[42];
	MM2VIS.rT_Cool_Air_Su	:=	rOpcVE_W[43];
	MM2VIS.rT_FreshAirEngA	:=	rOpcVE_W[44];
	MM2VIS.rT_FreshAirEngB	:=	rOpcVE_W[45];
	MM2VIS.rT_CircAirEng	:=	rOpcVE_W[46];
	MM2VIS.rT_AirER5		:=	rOpcVE_W[47];
	MM2VIS.rT_AirER6		:=	rOpcVE_W[48];

	Para.iVisRoomLou		:= REAL_TO_INT(rOpcVE_W[49]);
	Para.iNumInlLou			:= REAL_TO_INT(rOpcVE_W[50]);
	Para.iNumInlLouRoom		:= REAL_TO_INT(rOpcVE_W[51]);
	Para.iNumOutlLou		:= REAL_TO_INT(rOpcVE_W[52]);
	Para.iNumCircLou		:= REAL_TO_INT(rOpcVE_W[53]);
	Para.iNumInlLouEng		:= REAL_TO_INT(rOpcVE_W[54]);
	Para.iNumCircLouEng		:= REAL_TO_INT(rOpcVE_W[55]);
	Para.rTB_Cust[19]		:= rOpcVE_W[56]; (*visu: exchange generator/engine position*)

	Para.tCtr_IntakeAir.W_min	:=	rOpcVE_W[57];
	Para.tCtr_IntakeAir.W_max	:=	rOpcVE_W[58];

	MM2VIS.rT_HW_Air_Re_2	:=	rOpcVE_W[59];
	MM2VIS.rT_HW_Air_Su_2	:=	rOpcVE_W[60];
	MM2VIS.rT_Cool_Air_Re_2	:=	rOpcVE_W[61];
	MM2VIS.rT_Cool_Air_Su_2	:=	rOpcVE_W[62];
	MM2VIS.rT_HR_InAirCool_Su	:=	rOpcVE_W[63];
	MM2VIS.rT_HR_InAirCool_Re	:=	rOpcVE_W[64];
	MM2VIS.rCtr_HR_InAirCool	:=	rOpcVE_W[65];
	MM2VIS.rPos_InlLou3			:=	rOpcVE_W[66];
	MM2VIS.rPos_InlLou4			:=	rOpcVE_W[67];
	MM2VIS.rPos_InlLou5			:=	rOpcVE_W[68];
	MM2VIS.rPos_InlLou6			:=	rOpcVE_W[69];
	MM2VIS.rCtr_AuxRoom_Fan_FC	:= 	rOpcVE_W[70];
	MM2VIS.rT_AuxRoom			:=  rOpcVE_W[71];
	rOpcVE_W[72];
	rOpcVE_W[73];
	rOpcVE_W[74];
	rOpcVE_W[75];
	rOpcVE_W[76];
	rOpcVE_W[77];
	rOpcVE_W[78];
	rOpcVE_W[79];
	rOpcVE_W[80];

	(**BOOL**)
	MM2VIS.bInAirER_Fan1DemOn	:=	bOpcVE_W[0];
	MM2VIS.bOutAirER_Fan1DemOn	:=	bOpcVE_W[1];
	MM2VIS.bInAirEng_FanDemOn	:=	bOpcVE_W[2];
	MM2VIS.bDem_HeaterInAirEng	:=	bOpcVE_W[3];
	MM2VIS.bDem_PumpInAirEng	:=	bOpcVE_W[4];
	MM2VIS.bDem_EmptyInAirCool	:=	bOpcVE_W[5];
	MM2VIS.bTS_FrostProtection	:=	bOpcVE_W[6];
	MM2VIS.bDem_ERV_Aut_Exist	:=	bOpcVE_W[7];

	Para.bFreshAirEngAB_Active	:= bOpcVE_W[8];
	Para.bFB_AC_Heating_Active	:= bOpcVE_W[9];
	Para.bAirCondHeaterActive	:= bOpcVE_W[10];
	Para.bT_HW_Air_Re_Active	:= bOpcVE_W[11];
	Para.bPr_HW_Air_Re_Active	:= bOpcVE_W[12];
	Para.bT_HW_Air_Su_Active	:= bOpcVE_W[13];
	Para.bFB_AC_Cooling_Active	:= bOpcVE_W[14];
	Para.bT_Cool_Air_Re_Active	:= bOpcVE_W[15];
	Para.bPr_Cool_Air_Re_Active	:= bOpcVE_W[16];
	Para.bT_Cool_Air_Su_Active	:= bOpcVE_W[17];

	Para.bT_AirER1_Active		:= bOpcVE_W[18];
	Para.bT_AirER2_Active		:= bOpcVE_W[19];
	Para.bT_AirER3_Active		:= bOpcVE_W[20];
	Para.bT_AirER4_Active		:= bOpcVE_W[21];
	Para.bT_AirER5_Active		:= bOpcVE_W[22];
	Para.bT_AirER6_Active		:= bOpcVE_W[23];
	Para.bT_AirOutdoor_Active	:= bOpcVE_W[24];
	Para.bPrDiff_ER_Active		:= bOpcVE_W[25];
	Para.bCircLouActive			:= bOpcVE_W[26];
	Para.bCircLouEngActive		:= bOpcVE_W[27];
	Para.bT_CircAirEng_Active	:= bOpcVE_W[28];
	MM2VIS.bT_HW_Air_2_Active	:= bOpcVE_W[29];
	MM2VIS.bT_Cool_Air_2_Active := bOpcVE_W[30];

	MM2VIS.bDem_PumpInAirCool 	  := bOpcVE_W[31];
	MM2VIS.bDem_HR_CircPump_InAir := bOpcVE_W[32];
	MM2VIS.bAuxRoom_InLouOpened	  := bOpcVE_W[33];
	MM2VIS.bDem_Fan_AuxRoom		  := bOpcVE_W[34];
	bOpcVE_W[35];
	bOpcVE_W[36];
	bOpcVE_W[37];
	bOpcVE_W[38];
	bOpcVE_W[39];
	bOpcVE_W[40];

END_PROGRAM
```

### Program Logical/DataInterface/OpcMDE (IEC) - OPC Var for MDE
